LIN {X 0,Y 278.895,Z 532.06,A -85,B 0,C 180,E1 8838.94,E2 8838.94} C_VEL
LIN {X 0,Y 275.057,Z 524.837,A -85,B 0,C 180,E1 8835.829,E2 8835.829} C_VEL
LIN {X 0,Y 272.433,Z 520.123,A -85,B 0,C 180,E1 8833.269,E2 8833.269} C_VEL
LIN {X 0,Y 270.738,Z 517.123,A -85,B 0,C 180,E1 8831.296,E2 8831.296} C_VEL
LIN {X 0,Y 268.744,Z 513.445,A -85,B 0,C 180,E1 8828.352,E2 8828.352} C_VEL
LIN {X 0,Y 266.68,Z 509.32,A -85,B 0,C 180,E1 8823.018,E2 8823.018} C_VEL
LIN {X 0,Y 266.52,Z 508.712,A -85,B 0,C 180,E1 8821.944,E2 8821.944} C_VEL
LIN {X 0,Y 266.628,Z 508.877,A -85,B 0,C 180,E1 8817,E2 8817} C_VEL
LIN {X 0,Y 268.614,Z 513.288,A -85,B 0,C 180,E1 8811.447,E2 8811.447} C_VEL
LIN {X 0,Y 269.377,Z 514.72,A -85,B 0,C 180,E1 8810.179,E2 8810.179} C_VEL
LIN {X 0,Y 271.686,Z 518.794,A -85,B 0,C 180,E1 8807.145,E2 8807.145} C_VEL
LIN {X 0,Y 274.494,Z 523.834,A -85,B 0,C 180,E1 8804.265,E2 8804.265} C_VEL
LIN {X 0,Y 284.52,Z 539.001,A -85,B 0,C 180,E1 8797.161,E2 8797.161} C_VEL
LIN {X 0,Y 294.032,Z 548.26,A -85,B 0,C 180,E1 8792.575,E2 8792.575} C_VEL
LIN {X 0,Y 299.844,Z 552.837,A -85,B 0,C 180,E1 8790.22,E2 8790.22} C_VEL
LIN {X 0,Y 306.132,Z 557.593,A -85,B 0,C 180,E1 8787.514,E2 8787.514} C_VEL
LIN {X 0,Y 312.499,Z 562.998,A -85,B 0,C 180,E1 8784.512,E2 8784.512} C_VEL
LIN {X 0,Y 317.671,Z 567.158,A -85,B 0,C 180,E1 8781.808,E2 8781.808} C_VEL
LIN {X 0,Y 322.992,Z 572.197,A -85,B 0,C 180,E1 8778.644,E2 8778.644} C_VEL
LIN {X 0,Y 326.237,Z 574.988,A -85,B 0,C 180,E1 8776.659,E2 8776.659} C_VEL
LIN {X 0,Y 331.205,Z 579.653,A -85,B 0,C 180,E1 8773.494,E2 8773.494} C_VEL
LIN {X 0,Y 334.739,Z 582.505,A -85,B 0,C 180,E1 8771.19,E2 8771.19} C_VEL
LIN {X 0,Y 339.474,Z 587.061,A -85,B 0,C 180,E1 8767.893,E2 8767.893} C_VEL
LIN {X 0,Y 343.653,Z 590.222,A -85,B 0,C 180,E1 8764.886,E2 8764.886} C_VEL
LIN {X 0,Y 347.419,Z 593.994,A -85,B 0,C 180,E1 8761.917,E2 8761.917} C_VEL
LIN {X 0,Y 351.248,Z 596.825,A -85,B 0,C 180,E1 8758.755,E2 8758.755} C_VEL
LIN {X 0,Y 353.096,Z 598.088,A -85,B 0,C 180,E1 8757.122,E2 8757.122} C_VEL
LIN {X 0,Y 356.171,Z 601.48,A -85,B 0,C 180,E1 8754.019,E2 8754.019} C_VEL
LIN {X 0,Y 359.21,Z 603.908,A -85,B 0,C 180,E1 8750.701,E2 8750.701} C_VEL
LIN {X 0,Y 361.941,Z 605.377,A -85,B 0,C 180,E1 8747.358,E2 8747.358} C_VEL
LIN {X 0,Y 363.254,Z 606.183,A -85,B 0,C 180,E1 8745.485,E2 8745.485} C_VEL
LIN {X 0,Y 365.032,Z 608.588,A -85,B 0,C 180,E1 8742.336,E2 8742.336} C_VEL
LIN {X 0,Y 366.44,Z 610.11,A -85,B 0,C 180,E1 8739.05,E2 8739.05} C_VEL
LIN {X 0,Y 367.523,Z 611.035,A -85,B 0,C 180,E1 8735.62,E2 8735.62} C_VEL
LIN {X 0,Y 368.125,Z 611.482,A -85,B 0,C 180,E1 8732.179,E2 8732.179} C_VEL
LIN {X 0,Y 368.163,Z 611.49,A -85,B 0,C 180,E1 8728.911,E2 8728.911} C_VEL
LIN {X 0,Y 367.82,Z 611.243,A -85,B 0,C 180,E1 8725.635,E2 8725.635} C_VEL
LIN {X 0,Y 366.897,Z 610.529,A -85,B 0,C 180,E1 8722.169,E2 8722.169} C_VEL
LIN {X 0,Y 365.612,Z 609.266,A -85,B 0,C 180,E1 8718.964,E2 8718.964} C_VEL
LIN {X 0,Y 364.032,Z 607.268,A -85,B 0,C 180,E1 8715.782,E2 8715.782} C_VEL
LIN {X 0,Y 362.594,Z 605.615,A -85,B 0,C 180,E1 8713.5,E2 8713.5} C_VEL
LIN {X 0,Y 359.86,Z 604.308,A -85,B 0,C 180,E1 8710.017,E2 8710.017} C_VEL
LIN {X 0,Y 356.901,Z 602.129,A -85,B 0,C 180,E1 8706.734,E2 8706.734} C_VEL
LIN {X 0,Y 353.792,Z 598.981,A -85,B 0,C 180,E1 8703.597,E2 8703.597} C_VEL
LIN {X 0,Y 352.164,Z 597.33,A -85,B 0,C 180,E1 8702.066,E2 8702.066} C_VEL
LIN {X 0,Y 348.411,Z 594.838,A -85,B 0,C 180,E1 8698.899,E2 8698.899} C_VEL
LIN {X 0,Y 344.448,Z 591.117,A -85,B 0,C 180,E1 8695.728,E2 8695.728} C_VEL
LIN {X 0,Y 342.485,Z 589.191,A -85,B 0,C 180,E1 8694.234,E2 8694.234} C_VEL
LIN {X 0,Y 338.18,Z 585.932,A -85,B 0,C 180,E1 8691.187,E2 8691.187} C_VEL
LIN {X 0,Y 333.157,Z 581.089,A -85,B 0,C 180,E1 8687.76,E2 8687.76} C_VEL
LIN {X 0,Y 328.196,Z 577.001,A -85,B 0,C 180,E1 8684.579,E2 8684.579} C_VEL
LIN {X 0,Y 324.234,Z 573.152,A -85,B 0,C 180,E1 8682.108,E2 8682.108} C_VEL
LIN {X 0,Y 319.076,Z 568.633,A -85,B 0,C 180,E1 8679.026,E2 8679.026} C_VEL
LIN {X 0,Y 315.336,Z 565.145,A -85,B 0,C 180,E1 8676.919,E2 8676.919} C_VEL
LIN {X 0,Y 309.925,Z 560.861,A -85,B 0,C 180,E1 8674.248,E2 8674.248} C_VEL
LIN {X 0,Y 305.541,Z 557.19,A -85,B 0,C 180,E1 8672.223,E2 8672.223} C_VEL
LIN {X 0,Y 298.76,Z 551.933,A -85,B 0,C 180,E1 8669.348,E2 8669.348} C_VEL
LIN {X 0,Y 287.991,Z 542.764,A -85,B 0,C 180,E1 8664.665,E2 8664.665} C_VEL
LIN {X 0,Y 280.024,Z 533.138,A -85,B 0,C 180,E1 8660.09,E2 8660.09} C_VEL
LIN {X 0,Y 273.336,Z 521.624,A -85,B 0,C 180,E1 8654.609,E2 8654.609} C_VEL
LIN {X 0,Y 270.651,Z 517.002,A -85,B 0,C 180,E1 8651.605,E2 8651.605} C_VEL
LIN {X 0,Y 268.746,Z 513.415,A -85,B 0,C 180,E1 8648.764,E2 8648.764} C_VEL
LIN {X 0,Y 266.64,Z 508.986,A -85,B 0,C 180,E1 8643.107,E2 8643.107} C_VEL
LIN {X 0,Y 266.486,Z 508.701,A -85,B 0,C 180,E1 8638.271,E2 8638.271} C_VEL
LIN {X 0,Y 266.665,Z 509.22,A -85,B 0,C 180,E1 8637.089,E2 8637.089} C_VEL
LIN {X 0,Y 268.613,Z 513.317,A -85,B 0,C 180,E1 8631.86,E2 8631.86} C_VEL
LIN {X 0,Y 269.377,Z 514.737,A -85,B 0,C 180,E1 8630.592,E2 8630.592} C_VEL
LIN {X 0,Y 271.784,Z 518.909,A -85,B 0,C 180,E1 8627.456,E2 8627.456} C_VEL
LIN {X 0,Y 274.273,Z 523.465,A -85,B 0,C 180,E1 8624.883,E2 8624.883} C_VEL
LIN {X 0,Y 277.465,Z 529.282,A -85,B 0,C 180,E1 8622.155,E2 8622.155} C_VEL
LIN {X 0,Y 280.369,Z 535.335,A -85,B 0,C 180,E1 8619.972,E2 8619.972} C_VEL
LIN {X 0,Y 281.017,Z 537.508,A -85,B 0,C 180,E1 8619.462,E2 8619.462} C_VEL
LIN {X 0,Y 271.138,Z 641.697,A -85,B 0,C 180,E1 8617.288,E2 8617.288} C_VEL
LIN {X 0,Y 267.223,Z 664.526,A -85,B 0,C 180,E1 8616.63,E2 8616.63} C_VEL
LIN {X 0,Y 263.041,Z 681.531,A -85,B 0,C 180,E1 8615.964,E2 8615.964} C_VEL
LIN {X 0,Y 257.934,Z 698.333,A -85,B 0,C 180,E1 8615.101,E2 8615.101} C_VEL
LIN {X 0,Y 250.339,Z 718.684,A -85,B 0,C 180,E1 8613.719,E2 8613.719} C_VEL
LIN {X 0,Y 243.385,Z 734.31,A -85,B 0,C 180,E1 8612.331,E2 8612.331} C_VEL
LIN {X 0,Y 235.714,Z 749.491,A -85,B 0,C 180,E1 8610.653,E2 8610.653} C_VEL
LIN {X 0,Y 225.819,Z 766.74,A -85,B 0,C 180,E1 8608.222,E2 8608.222} C_VEL
LIN {X 0,Y 216.717,Z 780.747,A -85,B 0,C 180,E1 8605.672,E2 8605.672} C_VEL
LIN {X 0,Y 208.118,Z 792.952,A -85,B 0,C 180,E1 8602.891,E2 8602.891} C_VEL
LIN {X 0,Y 197.528,Z 806.818,A -85,B 0,C 180,E1 8598.836,E2 8598.836} C_VEL
LIN {X 0,Y 188.815,Z 817.411,A -85,B 0,C 180,E1 8594.771,E2 8594.771} C_VEL
LIN {X 0,Y 185.36,Z 821.62,A -85,B 0,C 180,E1 8592.894,E2 8592.894} C_VEL
LIN {X 0,Y 181.356,Z 825.4,A -85,B 0,C 180,E1 8591.182,E2 8591.182} C_VEL
LIN {X 0,Y 168.049,Z 834.548,A -85,B 0,C 180,E1 8586.633,E2 8586.633} C_VEL
LIN {X 0,Y 165.072,Z 837.01,A -85,B 0,C 180,E1 8584.778,E2 8584.778} C_VEL
LIN {X 0,Y 159.783,Z 842.971,A -85,B 0,C 180,E1 8579.214,E2 8579.214} C_VEL
LIN {X 0,Y 155.155,Z 848.829,A -85,B 0,C 180,E1 8571.846,E2 8571.846} C_VEL
LIN {X 0,Y 152.714,Z 852.655,A -85,B 0,C 180,E1 8564.406,E2 8564.406} C_VEL
LIN {X 0,Y 152.039,Z 854.633,A -85,B 0,C 180,E1 8558.318,E2 8558.318} C_VEL
LIN {X 0,Y 152.004,Z 855.505,A -85,B 0,C 180,E1 8553.016,E2 8553.016} C_VEL
LIN {X 0,Y 152.02,Z 855.596,A -85,B 0,C 180,E1 8548.115,E2 8548.115} C_VEL
LIN {X 0,Y 152.021,Z 854.815,A -85,B 0,C 180,E1 8542.442,E2 8542.442} C_VEL
LIN {X 0,Y 152.575,Z 852.957,A -85,B 0,C 180,E1 8536.355,E2 8536.355} C_VEL
LIN {X 0,Y 154.388,Z 849.835,A -85,B 0,C 180,E1 8529.926,E2 8529.926} C_VEL
LIN {X 0,Y 158.437,Z 844.654,A -85,B 0,C 180,E1 8522.57,E2 8522.57} C_VEL
LIN {X 0,Y 164.428,Z 837.72,A -85,B 0,C 180,E1 8515.812,E2 8515.812} C_VEL
LIN {X 0,Y 171.11,Z 830.424,A -85,B 0,C 180,E1 8510.438,E2 8510.438} C_VEL
LIN {X 0,Y 180.588,Z 820.031,A -85,B 0,C 180,E1 8504.696,E2 8504.696} C_VEL
LIN {X 0,Y 189.382,Z 809.898,A -85,B 0,C 180,E1 8500.509,E2 8500.509} C_VEL
LIN {X 0,Y 198.041,Z 799.411,A -85,B 0,C 180,E1 8497.091,E2 8497.091} C_VEL
LIN {X 0,Y 208.739,Z 785.512,A -85,B 0,C 180,E1 8493.547,E2 8493.547} C_VEL
LIN {X 0,Y 218.699,Z 770.992,A -85,B 0,C 180,E1 8490.741,E2 8490.741} C_VEL
LIN {X 0,Y 227.256,Z 757.259,A -85,B 0,C 180,E1 8488.633,E2 8488.633} C_VEL
LIN {X 0,Y 236.91,Z 739.862,A -85,B 0,C 180,E1 8486.53,E2 8486.53} C_VEL
LIN {X 0,Y 244.849,Z 723.051,A -85,B 0,C 180,E1 8484.971,E2 8484.971} C_VEL
LIN {X 0,Y 251.35,Z 707.199,A -85,B 0,C 180,E1 8483.808,E2 8483.808} C_VEL
LIN {X 0,Y 257.973,Z 688.057,A -85,B 0,C 180,E1 8482.718,E2 8482.718} C_VEL
LIN {X 0,Y 263.191,Z 668.401,A -85,B 0,C 180,E1 8481.912,E2 8481.912} C_VEL
LIN {X 0,Y 266.733,Z 650.8,A -85,B 0,C 180,E1 8481.37,E2 8481.37} C_VEL
LIN {X 0,Y 269.745,Z 627.11,A -85,B 0,C 180,E1 8480.812,E2 8480.812} C_VEL
LIN {X 0,Y 277.893,Z 541.402,A -85,B 0,C 180,E1 8479.066,E2 8479.066} C_VEL
LIN {X 0,Y 274.668,Z 534.689,A -85,B 0,C 180,E1 8476.449,E2 8476.449} C_VEL
LIN {X 0,Y 271.145,Z 527.997,A -85,B 0,C 180,E1 8473.008,E2 8473.008} C_VEL
LIN {X 0,Y 269.338,Z 524.692,A -85,B 0,C 180,E1 8470.814,E2 8470.814} C_VEL
LIN {X 0,Y 267.512,Z 521.194,A -85,B 0,C 180,E1 8467.958,E2 8467.958} C_VEL
LIN {X 0,Y 265.619,Z 516.917,A -85,B 0,C 180,E1 8462.49,E2 8462.49} C_VEL
LIN {X 0,Y 265.6,Z 516.697,A -85,B 0,C 180,E1 8457.312,E2 8457.312} C_VEL
LIN {X 0,Y 267.514,Z 521.166,A -85,B 0,C 180,E1 8451.628,E2 8451.628} C_VEL
LIN {X 0,Y 270.26,Z 526.374,A -85,B 0,C 180,E1 8447.599,E2 8447.599} C_VEL
LIN {X 0,Y 272.833,Z 531.197,A -85,B 0,C 180,E1 8444.82,E2 8444.82} C_VEL
LIN {X 0,Y 282.543,Z 546.368,A -85,B 0,C 180,E1 8437.652,E2 8437.652} C_VEL
LIN {X 0,Y 292.072,Z 555.804,A -85,B 0,C 180,E1 8432.927,E2 8432.927} C_VEL
LIN {X 0,Y 299.552,Z 561.757,A -85,B 0,C 180,E1 8429.857,E2 8429.857} C_VEL
LIN {X 0,Y 306.439,Z 566.905,A -85,B 0,C 180,E1 8426.884,E2 8426.884} C_VEL
LIN {X 0,Y 312.333,Z 571.835,A -85,B 0,C 180,E1 8424.038,E2 8424.038} C_VEL
LIN {X 0,Y 316.143,Z 574.926,A -85,B 0,C 180,E1 8422.051,E2 8422.051} C_VEL
LIN {X 0,Y 321.379,Z 579.816,A -85,B 0,C 180,E1 8418.984,E2 8418.984} C_VEL
LIN {X 0,Y 324.796,Z 582.75,A -85,B 0,C 180,E1 8416.904,E2 8416.904} C_VEL
LIN {X 0,Y 329.814,Z 587.419,A -85,B 0,C 180,E1 8413.724,E2 8413.724} C_VEL
LIN {X 0,Y 333.493,Z 590.415,A -85,B 0,C 180,E1 8411.336,E2 8411.336} C_VEL
LIN {X 0,Y 338.248,Z 594.926,A -85,B 0,C 180,E1 8408.04,E2 8408.04} C_VEL
LIN {X 0,Y 342.443,Z 598.118,A -85,B 0,C 180,E1 8405.034,E2 8405.034} C_VEL
LIN {X 0,Y 346.371,Z 601.979,A -85,B 0,C 180,E1 8401.952,E2 8401.952} C_VEL
LIN {X 0,Y 350.368,Z 604.862,A -85,B 0,C 180,E1 8398.647,E2 8398.647} C_VEL
LIN {X 0,Y 352.084,Z 606.158,A -85,B 0,C 180,E1 8397.123,E2 8397.123} C_VEL
LIN {X 0,Y 355.313,Z 609.596,A -85,B 0,C 180,E1 8393.884,E2 8393.884} C_VEL
LIN {X 0,Y 358.324,Z 611.937,A -85,B 0,C 180,E1 8390.584,E2 8390.584} C_VEL
LIN {X 0,Y 361.059,Z 613.362,A -85,B 0,C 180,E1 8387.216,E2 8387.216} C_VEL
LIN {X 0,Y 362.242,Z 614.145,A -85,B 0,C 180,E1 8385.529,E2 8385.529} C_VEL
LIN {X 0,Y 364.026,Z 616.531,A -85,B 0,C 180,E1 8382.371,E2 8382.371} C_VEL
LIN {X 0,Y 365.451,Z 618.049,A -85,B 0,C 180,E1 8379.073,E2 8379.073} C_VEL
LIN {X 0,Y 366.544,Z 618.975,A -85,B 0,C 180,E1 8375.635,E2 8375.635} C_VEL
LIN {X 0,Y 367.15,Z 619.423,A -85,B 0,C 180,E1 8372.185,E2 8372.185} C_VEL
LIN {X 0,Y 367.186,Z 619.43,A -85,B 0,C 180,E1 8368.908,E2 8368.908} C_VEL
LIN {X 0,Y 366.838,Z 619.182,A -85,B 0,C 180,E1 8365.623,E2 8365.623} C_VEL
LIN {X 0,Y 365.952,Z 618.516,A -85,B 0,C 180,E1 8362.306,E2 8362.306} C_VEL
LIN {X 0,Y 364.628,Z 617.227,A -85,B 0,C 180,E1 8358.96,E2 8358.96} C_VEL
LIN {X 0,Y 363.031,Z 615.245,A -85,B 0,C 180,E1 8355.763,E2 8355.763} C_VEL
LIN {X 0,Y 361.57,Z 613.544,A -85,B 0,C 180,E1 8353.452,E2 8353.452} C_VEL
LIN {X 0,Y 358.972,Z 612.321,A -85,B 0,C 180,E1 8350.135,E2 8350.135} C_VEL
LIN {X 0,Y 356.011,Z 610.204,A -85,B 0,C 180,E1 8346.848,E2 8346.848} C_VEL
LIN {X 0,Y 352.767,Z 607.007,A -85,B 0,C 180,E1 8343.578,E2 8343.578} C_VEL
LIN {X 0,Y 351.056,Z 605.231,A -85,B 0,C 180,E1 8341.97,E2 8341.97} C_VEL
LIN {X 0,Y 347.231,Z 602.709,A -85,B 0,C 180,E1 8338.763,E2 8338.763} C_VEL
LIN {X 0,Y 343.157,Z 598.927,A -85,B 0,C 180,E1 8335.527,E2 8335.527} C_VEL
LIN {X 0,Y 340.974,Z 596.877,A -85,B 0,C 180,E1 8333.887,E2 8333.887} C_VEL
LIN {X 0,Y 336.485,Z 593.404,A -85,B 0,C 180,E1 8330.735,E2 8330.735} C_VEL
LIN {X 0,Y 331.805,Z 588.879,A -85,B 0,C 180,E1 8327.548,E2 8327.548} C_VEL
LIN {X 0,Y 326.77,Z 584.766,A -85,B 0,C 180,E1 8324.346,E2 8324.346} C_VEL
LIN {X 0,Y 322.635,Z 580.784,A -85,B 0,C 180,E1 8321.768,E2 8321.768} C_VEL
LIN {X 0,Y 317.419,Z 576.231,A -85,B 0,C 180,E1 8318.688,E2 8318.688} C_VEL
LIN {X 0,Y 313.764,Z 572.877,A -85,B 0,C 180,E1 8316.678,E2 8316.678} C_VEL
LIN {X 0,Y 308.135,Z 568.446,A -85,B 0,C 180,E1 8313.913,E2 8313.913} C_VEL
LIN {X 0,Y 303.304,Z 564.494,A -85,B 0,C 180,E1 8311.71,E2 8311.71} C_VEL
LIN {X 0,Y 296.567,Z 559.304,A -85,B 0,C 180,E1 8308.922,E2 8308.922} C_VEL
LIN {X 0,Y 286.028,Z 550.228,A -85,B 0,C 180,E1 8304.24,E2 8304.24} C_VEL
LIN {X 0,Y 278.095,Z 540.397,A -85,B 0,C 180,E1 8299.523,E2 8299.523} C_VEL
LIN {X 0,Y 271.724,Z 529.017,A -85,B 0,C 180,E1 8294.045,E2 8294.045} C_VEL
LIN {X 0,Y 269.337,Z 524.691,A -85,B 0,C 180,E1 8291.228,E2 8291.228} C_VEL
LIN {X 0,Y 267.514,Z 521.166,A -85,B 0,C 180,E1 8288.372,E2 8288.372} C_VEL
LIN {X 0,Y 265.545,Z 516.653,A -85,B 0,C 180,E1 8282.364,E2 8282.364} C_VEL
LIN {X 0,Y 265.619,Z 516.917,A -85,B 0,C 180,E1 8277.51,E2 8277.51} C_VEL
LIN {X 0,Y 267.512,Z 521.194,A -85,B 0,C 180,E1 8272.042,E2 8272.042} C_VEL
LIN {X 0,Y 270.337,Z 526.453,A -85,B 0,C 180,E1 8267.93,E2 8267.93} C_VEL
LIN {X 0,Y 272.936,Z 531.424,A -85,B 0,C 180,E1 8265.133,E2 8265.133} C_VEL
LIN {X 0,Y 276.109,Z 537.585,A -85,B 0,C 180,E1 8262.337,E2 8262.337} C_VEL
LIN {X 0,Y 277.894,Z 541.512,A -85,B 0,C 180,E1 8260.926,E2 8260.926} C_VEL
LIN {X 0,Y 268.116,Z 641.667,A -85,B 0,C 180,E1 8258.866,E2 8258.866} C_VEL
LIN {X 0,Y 264.072,Z 664.592,A -85,B 0,C 180,E1 8258.217,E2 8258.217} C_VEL
LIN {X 0,Y 259.921,Z 681.125,A -85,B 0,C 180,E1 8257.589,E2 8257.589} C_VEL
LIN {X 0,Y 255.021,Z 696.98,A -85,B 0,C 180,E1 8256.805,E2 8256.805} C_VEL
LIN {X 0,Y 248.096,Z 715.668,A -85,B 0,C 180,E1 8255.613,E2 8255.613} C_VEL
LIN {X 0,Y 240.061,Z 733.408,A -85,B 0,C 180,E1 8254.108,E2 8254.108} C_VEL
LIN {X 0,Y 232.621,Z 747.828,A -85,B 0,C 180,E1 8252.568,E2 8252.568} C_VEL
LIN {X 0,Y 223.504,Z 763.57,A -85,B 0,C 180,E1 8250.468,E2 8250.468} C_VEL
LIN {X 0,Y 212.932,Z 779.505,A -85,B 0,C 180,E1 8247.693,E2 8247.693} C_VEL
LIN {X 0,Y 203.957,Z 791.818,A -85,B 0,C 180,E1 8244.951,E2 8244.951} C_VEL
LIN {X 0,Y 193.631,Z 804.96,A -85,B 0,C 180,E1 8241.233,E2 8241.233} C_VEL
LIN {X 0,Y 183.632,Z 816.547,A -85,B 0,C 180,E1 8236.853,E2 8236.853} C_VEL
LIN {X 0,Y 175.782,Z 825.3,A -85,B 0,C 180,E1 8232.599,E2 8232.599} C_VEL
LIN {X 0,Y 167.551,Z 834.392,A -85,B 0,C 180,E1 8226.885,E2 8226.885} C_VEL
LIN {X 0,Y 165.072,Z 837.01,A -85,B 0,C 180,E1 8224.778,E2 8224.778} C_VEL
LIN {X 0,Y 161.674,Z 839.89,A -85,B 0,C 180,E1 8222.527,E2 8222.527} C_VEL
LIN {X 0,Y 150.726,Z 845.91,A -85,B 0,C 180,E1 8216.73,E2 8216.73} C_VEL
LIN {X 0,Y 148.111,Z 847.909,A -85,B 0,C 180,E1 8214.037,E2 8214.037} C_VEL
LIN {X 0,Y 144.945,Z 852.263,A -85,B 0,C 180,E1 8205.606,E2 8205.606} C_VEL
LIN {X 0,Y 144.077,Z 854.304,A -85,B 0,C 180,E1 8199.184,E2 8199.184} C_VEL
LIN {X 0,Y 143.999,Z 855.237,A -85,B 0,C 180,E1 8193.583,E2 8193.583} C_VEL
LIN {X 0,Y 144.027,Z 855.389,A -85,B 0,C 180,E1 8188.409,E2 8188.409} C_VEL
LIN {X 0,Y 144.023,Z 854.668,A -85,B 0,C 180,E1 8182.421,E2 8182.421} C_VEL
LIN {X 0,Y 144.62,Z 852.868,A -85,B 0,C 180,E1 8175.997,E2 8175.997} C_VEL
LIN {X 0,Y 146.602,Z 849.772,A -85,B 0,C 180,E1 8169.163,E2 8169.163} C_VEL
LIN {X 0,Y 150.925,Z 844.72,A -85,B 0,C 180,E1 8161.512,E2 8161.512} C_VEL
LIN {X 0,Y 157.539,Z 837.642,A -85,B 0,C 180,E1 8154.276,E2 8154.276} C_VEL
LIN {X 0,Y 164.384,Z 830.652,A -85,B 0,C 180,E1 8148.937,E2 8148.937} C_VEL
LIN {X 0,Y 173.581,Z 821.245,A -85,B 0,C 180,E1 8143.468,E2 8143.468} C_VEL
LIN {X 0,Y 183.673,Z 810.21,A -85,B 0,C 180,E1 8138.772,E2 8138.772} C_VEL
LIN {X 0,Y 192.546,Z 799.963,A -85,B 0,C 180,E1 8135.388,E2 8135.388} C_VEL
LIN {X 0,Y 202.909,Z 787.117,A -85,B 0,C 180,E1 8132.057,E2 8132.057} C_VEL
LIN {X 0,Y 213.899,Z 771.874,A -85,B 0,C 180,E1 8129.062,E2 8129.062} C_VEL
LIN {X 0,Y 222.712,Z 758.259,A -85,B 0,C 180,E1 8126.975,E2 8126.975} C_VEL
LIN {X 0,Y 231.396,Z 743.318,A -85,B 0,C 180,E1 8125.147,E2 8125.147} C_VEL
LIN {X 0,Y 240.729,Z 724.655,A -85,B 0,C 180,E1 8123.381,E2 8123.381} C_VEL
LIN {X 0,Y 247.369,Z 709.087,A -85,B 0,C 180,E1 8122.244,E2 8122.244} C_VEL
LIN {X 0,Y 253.321,Z 692.741,A -85,B 0,C 180,E1 8121.301,E2 8121.301} C_VEL
LIN {X 0,Y 259.399,Z 672.025,A -85,B 0,C 180,E1 8120.405,E2 8120.405} C_VEL
LIN {X 0,Y 263.411,Z 653.366,A -85,B 0,C 180,E1 8119.824,E2 8119.824} C_VEL
LIN {X 0,Y 266.081,Z 635.287,A -85,B 0,C 180,E1 8119.381,E2 8119.381} C_VEL
LIN {X 0,Y 274.883,Z 546.094,A -85,B 0,C 180,E1 8117.58,E2 8117.58} C_VEL
LIN {X 0,Y 271.501,Z 539.175,A -85,B 0,C 180,E1 8114.511,E2 8114.511} C_VEL
LIN {X 0,Y 268.909,Z 533.998,A -85,B 0,C 180,E1 8111.591,E2 8111.591} C_VEL
LIN {X 0,Y 266.292,Z 528.944,A -85,B 0,C 180,E1 8107.56,E2 8107.56} C_VEL
LIN {X 0,Y 264.537,Z 524.582,A -85,B 0,C 180,E1 8101.742,E2 8101.742} C_VEL
LIN {X 0,Y 264.606,Z 524.804,A -85,B 0,C 180,E1 8097.302,E2 8097.302} C_VEL
LIN {X 0,Y 266.7,Z 529.664,A -85,B 0,C 180,E1 8091.277,E2 8091.277} C_VEL
LIN {X 0,Y 268.901,Z 534.069,A -85,B 0,C 180,E1 8087.992,E2 8087.992} C_VEL
LIN {X 0,Y 271.611,Z 539.341,A -85,B 0,C 180,E1 8084.969,E2 8084.969} C_VEL
LIN {X 0,Y 280.586,Z 553.734,A -85,B 0,C 180,E1 8078.149,E2 8078.149} C_VEL
LIN {X 0,Y 290.123,Z 563.348,A -85,B 0,C 180,E1 8073.284,E2 8073.284} C_VEL
LIN {X 0,Y 299.893,Z 571.038,A -85,B 0,C 180,E1 8069.23,E2 8069.23} C_VEL
LIN {X 0,Y 304.96,Z 574.839,A -85,B 0,C 180,E1 8067.039,E2 8067.039} C_VEL
LIN {X 0,Y 310.954,Z 579.702,A -85,B 0,C 180,E1 8064.195,E2 8064.195} C_VEL
LIN {X 0,Y 314.779,Z 582.857,A -85,B 0,C 180,E1 8062.204,E2 8062.204} C_VEL
LIN {X 0,Y 320.154,Z 587.745,A -85,B 0,C 180,E1 8059.091,E2 8059.091} C_VEL
LIN {X 0,Y 323.405,Z 590.571,A -85,B 0,C 180,E1 8057.113,E2 8057.113} C_VEL
LIN {X 0,Y 328.428,Z 595.184,A -85,B 0,C 180,E1 8053.955,E2 8053.955} C_VEL
LIN {X 0,Y 332.099,Z 598.164,A -85,B 0,C 180,E1 8051.584,E2 8051.584} C_VEL
LIN {X 0,Y 336.809,Z 602.61,A -85,B 0,C 180,E1 8048.347,E2 8048.347} C_VEL
LIN {X 0,Y 341.134,Z 605.891,A -85,B 0,C 180,E1 8045.267,E2 8045.267} C_VEL
LIN {X 0,Y 345.186,Z 609.843,A -85,B 0,C 180,E1 8042.102,E2 8042.102} C_VEL
LIN {X 0,Y 349.16,Z 612.707,A -85,B 0,C 180,E1 8038.827,E2 8038.827} C_VEL
LIN {X 0,Y 350.902,Z 614.029,A -85,B 0,C 180,E1 8037.274,E2 8037.274} C_VEL
LIN {X 0,Y 354.015,Z 617.333,A -85,B 0,C 180,E1 8034.174,E2 8034.174} C_VEL
LIN {X 0,Y 357.148,Z 619.775,A -85,B 0,C 180,E1 8030.794,E2 8030.794} C_VEL
LIN {X 0,Y 359.903,Z 621.234,A -85,B 0,C 180,E1 8027.459,E2 8027.459} C_VEL
LIN {X 0,Y 361.209,Z 622.074,A -85,B 0,C 180,E1 8025.612,E2 8025.612} C_VEL
LIN {X 0,Y 363.02,Z 624.473,A -85,B 0,C 180,E1 8022.405,E2 8022.405} C_VEL
LIN {X 0,Y 364.439,Z 625.97,A -85,B 0,C 180,E1 8019.156,E2 8019.156} C_VEL
LIN {X 0,Y 365.537,Z 626.883,A -85,B 0,C 180,E1 8015.808,E2 8015.808} C_VEL
LIN {X 0,Y 366.126,Z 627.328,A -85,B 0,C 180,E1 8012.504,E2 8012.504} C_VEL
LIN {X 0,Y 366.216,Z 627.381,A -85,B 0,C 180,E1 8009.061,E2 8009.061} C_VEL
LIN {X 0,Y 365.893,Z 627.139,A -85,B 0,C 180,E1 8005.733,E2 8005.733} C_VEL
LIN {X 0,Y 365.009,Z 626.499,A -85,B 0,C 180,E1 8002.445,E2 8002.445} C_VEL
LIN {X 0,Y 363.695,Z 625.245,A -85,B 0,C 180,E1 7999.065,E2 7999.065} C_VEL
LIN {X 0,Y 362.049,Z 623.242,A -85,B 0,C 180,E1 7995.772,E2 7995.772} C_VEL
LIN {X 0,Y 360.546,Z 621.473,A -85,B 0,C 180,E1 7993.404,E2 7993.404} C_VEL
LIN {X 0,Y 357.938,Z 620.246,A -85,B 0,C 180,E1 7990.075,E2 7990.075} C_VEL
LIN {X 0,Y 354.871,Z 618.058,A -85,B 0,C 180,E1 7986.682,E2 7986.682} C_VEL
LIN {X 0,Y 351.675,Z 614.949,A -85,B 0,C 180,E1 7983.49,E2 7983.49} C_VEL
LIN {X 0,Y 349.716,Z 613.015,A -85,B 0,C 180,E1 7981.667,E2 7981.667} C_VEL
LIN {X 0,Y 345.836,Z 610.404,A -85,B 0,C 180,E1 7978.447,E2 7978.447} C_VEL
LIN {X 0,Y 341.728,Z 606.579,A -85,B 0,C 180,E1 7975.213,E2 7975.213} C_VEL
LIN {X 0,Y 339.736,Z 604.724,A -85,B 0,C 180,E1 7973.727,E2 7973.727} C_VEL
LIN {X 0,Y 335.2,Z 601.239,A -85,B 0,C 180,E1 7970.555,E2 7970.555} C_VEL
LIN {X 0,Y 330.273,Z 596.544,A -85,B 0,C 180,E1 7967.219,E2 7967.219} C_VEL
LIN {X 0,Y 325.137,Z 592.331,A -85,B 0,C 180,E1 7963.981,E2 7963.981} C_VEL
LIN {X 0,Y 321.185,Z 588.529,A -85,B 0,C 180,E1 7961.521,E2 7961.521} C_VEL
LIN {X 0,Y 315.938,Z 583.988,A -85,B 0,C 180,E1 7958.439,E2 7958.439} C_VEL
LIN {X 0,Y 312.015,Z 580.484,A -85,B 0,C 180,E1 7956.346,E2 7956.346} C_VEL
LIN {X 0,Y 306.139,Z 575.864,A -85,B 0,C 180,E1 7953.489,E2 7953.489} C_VEL
LIN {X 0,Y 301.371,Z 572.062,A -85,B 0,C 180,E1 7951.379,E2 7951.379} C_VEL
LIN {X 0,Y 294.58,Z 566.858,A -85,B 0,C 180,E1 7948.581,E2 7948.581} C_VEL
LIN {X 0,Y 283.992,Z 557.591,A -85,B 0,C 180,E1 7943.762,E2 7943.762} C_VEL
LIN {X 0,Y 276.194,Z 547.655,A -85,B 0,C 180,E1 7938.949,E2 7938.949} C_VEL
LIN {X 0,Y 270.237,Z 536.562,A -85,B 0,C 180,E1 7933.578,E2 7933.578} C_VEL
LIN {X 0,Y 267.957,Z 532.259,A -85,B 0,C 180,E1 7930.742,E2 7930.742} C_VEL
LIN {X 0,Y 266.295,Z 528.914,A -85,B 0,C 180,E1 7927.976,E2 7927.976} C_VEL
LIN {X 0,Y 264.537,Z 524.576,A -85,B 0,C 180,E1 7922.157,E2 7922.157} C_VEL
LIN {X 0,Y 264.604,Z 524.819,A -85,B 0,C 180,E1 7917.717,E2 7917.717} C_VEL
LIN {X 0,Y 266.413,Z 529.072,A -85,B 0,C 180,E1 7912.226,E2 7912.226} C_VEL
LIN {X 0,Y 268.991,Z 534.175,A -85,B 0,C 180,E1 7908.304,E2 7908.304} C_VEL
LIN {X 0,Y 271.606,Z 539.367,A -85,B 0,C 180,E1 7905.386,E2 7905.386} C_VEL
LIN {X 0,Y 274.891,Z 546.109,A -85,B 0,C 180,E1 7902.414,E2 7902.414} C_VEL
LIN {X 0,Y 265.328,Z 641.44,A -85,B 0,C 180,E1 7900.482,E2 7900.482} C_VEL
LIN {X 0,Y 261.219,Z 664.273,A -85,B 0,C 180,E1 7899.855,E2 7899.855} C_VEL
LIN {X 0,Y 256.896,Z 681.129,A -85,B 0,C 180,E1 7899.235,E2 7899.235} C_VEL
LIN {X 0,Y 251.581,Z 697.858,A -85,B 0,C 180,E1 7898.428,E2 7898.428} C_VEL
LIN {X 0,Y 243.623,Z 718.207,A -85,B 0,C 180,E1 7897.124,E2 7897.124} C_VEL
LIN {X 0,Y 236.234,Z 733.976,A -85,B 0,C 180,E1 7895.794,E2 7895.794} C_VEL
LIN {X 0,Y 228.206,Z 749.012,A -85,B 0,C 180,E1 7894.204,E2 7894.204} C_VEL
LIN {X 0,Y 217.692,Z 766.259,A -85,B 0,C 180,E1 7891.864,E2 7891.864} C_VEL
LIN {X 0,Y 207.955,Z 780.265,A -85,B 0,C 180,E1 7889.386,E2 7889.386} C_VEL
LIN {X 0,Y 198.679,Z 792.469,A -85,B 0,C 180,E1 7886.655,E2 7886.655} C_VEL
LIN {X 0,Y 187.318,Z 806.144,A -85,B 0,C 180,E1 7882.684,E2 7882.684} C_VEL
LIN {X 0,Y 177.536,Z 816.926,A -85,B 0,C 180,E1 7878.505,E2 7878.505} C_VEL
LIN {X 0,Y 168.793,Z 826.145,A -85,B 0,C 180,E1 7873.871,E2 7873.871} C_VEL
LIN {X 0,Y 159.126,Z 836.032,A -85,B 0,C 180,E1 7867.099,E2 7867.099} C_VEL
LIN {X 0,Y 152.975,Z 842.397,A -85,B 0,C 180,E1 7861.079,E2 7861.079} C_VEL
LIN {X 0,Y 148.111,Z 847.909,A -85,B 0,C 180,E1 7854.037,E2 7854.037} C_VEL
LIN {X 0,Y 145.773,Z 849.751,A -85,B 0,C 180,E1 7851.241,E2 7851.241} C_VEL
LIN {X 0,Y 139.583,Z 852.307,A -85,B 0,C 180,E1 7846.042,E2 7846.042} C_VEL
LIN {X 0,Y 136.526,Z 853.559,A -85,B 0,C 180,E1 7842.084,E2 7842.084} C_VEL
LIN {X 0,Y 136.181,Z 853.858,A -85,B 0,C 180,E1 7840.69,E2 7840.69} C_VEL
LIN {X 0,Y 135.995,Z 854.969,A -85,B 0,C 180,E1 7834.216,E2 7834.216} C_VEL
LIN {X 0,Y 136.028,Z 855.153,A -85,B 0,C 180,E1 7828.315,E2 7828.315} C_VEL
LIN {X 0,Y 136.035,Z 854.43,A -85,B 0,C 180,E1 7821.973,E2 7821.973} C_VEL
LIN {X 0,Y 136.835,Z 852.476,A -85,B 0,C 180,E1 7814.747,E2 7814.747} C_VEL
LIN {X 0,Y 139.15,Z 849.352,A -85,B 0,C 180,E1 7807.616,E2 7807.616} C_VEL
LIN {X 0,Y 144.325,Z 843.889,A -85,B 0,C 180,E1 7799.237,E2 7799.237} C_VEL
LIN {X 0,Y 150.942,Z 837.399,A -85,B 0,C 180,E1 7792.454,E2 7792.454} C_VEL
LIN {X 0,Y 158.277,Z 830.409,A -85,B 0,C 180,E1 7786.982,E2 7786.982} C_VEL
LIN {X 0,Y 168.452,Z 820.588,A -85,B 0,C 180,E1 7781.228,E2 7781.228} C_VEL
LIN {X 0,Y 179.159,Z 809.422,A -85,B 0,C 180,E1 7776.523,E2 7776.523} C_VEL
LIN {X 0,Y 188.762,Z 798.771,A -85,B 0,C 180,E1 7773.078,E2 7773.078} C_VEL
LIN {X 0,Y 200.548,Z 784.529,A -85,B 0,C 180,E1 7769.545,E2 7769.545} C_VEL
LIN {X 0,Y 210.841,Z 770.51,A -85,B 0,C 180,E1 7766.936,E2 7766.936} C_VEL
LIN {X 0,Y 219.936,Z 756.778,A -85,B 0,C 180,E1 7764.916,E2 7764.916} C_VEL
LIN {X 0,Y 230.134,Z 739.384,A -85,B 0,C 180,E1 7762.921,E2 7762.921} C_VEL
LIN {X 0,Y 238.481,Z 722.574,A -85,B 0,C 180,E1 7761.451,E2 7761.451} C_VEL
LIN {X 0,Y 245.288,Z 706.723,A -85,B 0,C 180,E1 7760.362,E2 7760.362} C_VEL
LIN {X 0,Y 252.198,Z 687.582,A -85,B 0,C 180,E1 7759.345,E2 7759.345} C_VEL
LIN {X 0,Y 257.65,Z 667.846,A -85,B 0,C 180,E1 7758.596,E2 7758.596} C_VEL
LIN {X 0,Y 261.32,Z 650.282,A -85,B 0,C 180,E1 7758.089,E2 7758.089} C_VEL
LIN {X 0,Y 264.493,Z 626.381,A -85,B 0,C 180,E1 7757.555,E2 7757.555} C_VEL
LIN {X 0,Y 272.032,Z 551.115,A -85,B 0,C 180,E1 7756.071,E2 7756.071} C_VEL
LIN {X 0,Y 269.12,Z 544.927,A -85,B 0,C 180,E1 7753.107,E2 7753.107} C_VEL
LIN {X 0,Y 266.743,Z 540.068,A -85,B 0,C 180,E1 7750.047,E2 7750.047} C_VEL
LIN {X 0,Y 265.085,Z 536.691,A -85,B 0,C 180,E1 7747.159,E2 7747.159} C_VEL
LIN {X 0,Y 263.531,Z 532.515,A -85,B 0,C 180,E1 7741.531,E2 7741.531} C_VEL
LIN {X 0,Y 263.595,Z 532.71,A -85,B 0,C 180,E1 7737.51,E2 7737.51} C_VEL
LIN {X 0,Y 265.529,Z 537.508,A -85,B 0,C 180,E1 7731.565,E2 7731.565} C_VEL
LIN {X 0,Y 267.571,Z 541.792,A -85,B 0,C 180,E1 7728.369,E2 7728.369} C_VEL
LIN {X 0,Y 270.186,Z 547.087,A -85,B 0,C 180,E1 7725.326,E2 7725.326} C_VEL
LIN {X 0,Y 278.493,Z 560.915,A -85,B 0,C 180,E1 7718.75,E2 7718.75} C_VEL
LIN {X 0,Y 288.186,Z 570.892,A -85,B 0,C 180,E1 7713.646,E2 7713.646} C_VEL
LIN {X 0,Y 298.596,Z 579.047,A -85,B 0,C 180,E1 7709.305,E2 7709.305} C_VEL
LIN {X 0,Y 303.288,Z 582.592,A -85,B 0,C 180,E1 7707.284,E2 7707.284} C_VEL
LIN {X 0,Y 309.187,Z 587.299,A -85,B 0,C 180,E1 7704.529,E2 7704.529} C_VEL
LIN {X 0,Y 313.245,Z 590.618,A -85,B 0,C 180,E1 7702.448,E2 7702.448} C_VEL
LIN {X 0,Y 318.537,Z 595.368,A -85,B 0,C 180,E1 7699.428,E2 7699.428} C_VEL
LIN {X 0,Y 321.908,Z 598.272,A -85,B 0,C 180,E1 7697.396,E2 7697.396} C_VEL
LIN {X 0,Y 327.152,Z 603.045,A -85,B 0,C 180,E1 7694.108,E2 7694.108} C_VEL
LIN {X 0,Y 330.68,Z 605.915,A -85,B 0,C 180,E1 7691.829,E2 7691.829} C_VEL
LIN {X 0,Y 335.659,Z 610.537,A -85,B 0,C 180,E1 7688.442,E2 7688.442} C_VEL
LIN {X 0,Y 339.915,Z 613.789,A -85,B 0,C 180,E1 7685.412,E2 7685.412} C_VEL
LIN {X 0,Y 343.974,Z 617.699,A -85,B 0,C 180,E1 7682.254,E2 7682.254} C_VEL
LIN {X 0,Y 347.871,Z 620.513,A -85,B 0,C 180,E1 7679.06,E2 7679.06} C_VEL
LIN {X 0,Y 349.635,Z 621.803,A -85,B 0,C 180,E1 7677.504,E2 7677.504} C_VEL
LIN {X 0,Y 352.967,Z 625.284,A -85,B 0,C 180,E1 7674.224,E2 7674.224} C_VEL
LIN {X 0,Y 356.137,Z 627.722,A -85,B 0,C 180,E1 7670.819,E2 7670.819} C_VEL
LIN {X 0,Y 358.884,Z 629.163,A -85,B 0,C 180,E1 7667.511,E2 7667.511} C_VEL
LIN {X 0,Y 360.13,Z 629.924,A -85,B 0,C 180,E1 7665.788,E2 7665.788} C_VEL
LIN {X 0,Y 361.913,Z 632.322,A -85,B 0,C 180,E1 7662.606,E2 7662.606} C_VEL
LIN {X 0,Y 363.388,Z 633.861,A -85,B 0,C 180,E1 7659.342,E2 7659.342} C_VEL
LIN {X 0,Y 364.501,Z 634.753,A -85,B 0,C 180,E1 7656.141,E2 7656.141} C_VEL
LIN {X 0,Y 365.092,Z 635.229,A -85,B 0,C 180,E1 7652.825,E2 7652.825} C_VEL
LIN {X 0,Y 365.26,Z 635.352,A -85,B 0,C 180,E1 7649.373,E2 7649.373} C_VEL
LIN {X 0,Y 364.973,Z 635.125,A -85,B 0,C 180,E1 7646.073,E2 7646.073} C_VEL
LIN {X 0,Y 364.114,Z 634.513,A -85,B 0,C 180,E1 7642.743,E2 7642.743} C_VEL
LIN {X 0,Y 362.86,Z 633.355,A -85,B 0,C 180,E1 7639.361,E2 7639.361} C_VEL
LIN {X 0,Y 361.225,Z 631.454,A -85,B 0,C 180,E1 7636.066,E2 7636.066} C_VEL
LIN {X 0,Y 359.523,Z 629.402,A -85,B 0,C 180,E1 7633.355,E2 7633.355} C_VEL
LIN {X 0,Y 356.9,Z 628.17,A -85,B 0,C 180,E1 7630.015,E2 7630.015} C_VEL
LIN {X 0,Y 353.855,Z 626.019,A -85,B 0,C 180,E1 7626.655,E2 7626.655} C_VEL
LIN {X 0,Y 350.584,Z 622.889,A -85,B 0,C 180,E1 7623.401,E2 7623.401} C_VEL
LIN {X 0,Y 348.612,Z 620.916,A -85,B 0,C 180,E1 7621.57,E2 7621.57} C_VEL
LIN {X 0,Y 344.688,Z 618.297,A -85,B 0,C 180,E1 7618.33,E2 7618.33} C_VEL
LIN {X 0,Y 340.528,Z 614.478,A -85,B 0,C 180,E1 7615.072,E2 7615.072} C_VEL
LIN {X 0,Y 338.37,Z 612.486,A -85,B 0,C 180,E1 7613.471,E2 7613.471} C_VEL
LIN {X 0,Y 333.834,Z 608.994,A -85,B 0,C 180,E1 7610.313,E2 7610.313} C_VEL
LIN {X 0,Y 328.859,Z 604.296,A -85,B 0,C 180,E1 7606.973,E2 7606.973} C_VEL
LIN {X 0,Y 323.608,Z 599.987,A -85,B 0,C 180,E1 7603.672,E2 7603.672} C_VEL
LIN {X 0,Y 319.57,Z 596.156,A -85,B 0,C 180,E1 7601.18,E2 7601.18} C_VEL
LIN {X 0,Y 314.256,Z 591.586,A -85,B 0,C 180,E1 7598.102,E2 7598.102} C_VEL
LIN {X 0,Y 310.1,Z 587.961,A -85,B 0,C 180,E1 7595.919,E2 7595.919} C_VEL
LIN {X 0,Y 303.879,Z 583.107,A -85,B 0,C 180,E1 7592.981,E2 7592.981} C_VEL
LIN {X 0,Y 299.435,Z 579.628,A -85,B 0,C 180,E1 7591.045,E2 7591.045} C_VEL
LIN {X 0,Y 292.369,Z 574.223,A -85,B 0,C 180,E1 7588.148,E2 7588.148} C_VEL
LIN {X 0,Y 282.063,Z 565.053,A -85,B 0,C 180,E1 7583.325,E2 7583.325} C_VEL
LIN {X 0,Y 274.322,Z 554.913,A -85,B 0,C 180,E1 7578.367,E2 7578.367} C_VEL
LIN {X 0,Y 268.675,Z 543.952,A -85,B 0,C 180,E1 7573.001,E2 7573.001} C_VEL
LIN {X 0,Y 266.526,Z 539.7,A -85,B 0,C 180,E1 7570.145,E2 7570.145} C_VEL
LIN {X 0,Y 265.09,Z 536.659,A -85,B 0,C 180,E1 7567.576,E2 7567.576} C_VEL
LIN {X 0,Y 263.533,Z 532.5,A -85,B 0,C 180,E1 7561.947,E2 7561.947} C_VEL
LIN {X 0,Y 263.586,Z 532.618,A -85,B 0,C 180,E1 7558.034,E2 7558.034} C_VEL
LIN {X 0,Y 265.527,Z 537.52,A -85,B 0,C 180,E1 7551.982,E2 7551.982} C_VEL
LIN {X 0,Y 267.656,Z 541.894,A -85,B 0,C 180,E1 7548.681,E2 7548.681} C_VEL
LIN {X 0,Y 270.489,Z 547.695,A -85,B 0,C 180,E1 7545.433,E2 7545.433} C_VEL
LIN {X 0,Y 272.022,Z 551.376,A -85,B 0,C 180,E1 7543.912,E2 7543.912} C_VEL
LIN {X 0,Y 262.73,Z 641.41,A -85,B 0,C 180,E1 7542.127,E2 7542.127} C_VEL
LIN {X 0,Y 258.538,Z 664.151,A -85,B 0,C 180,E1 7541.521,E2 7541.521} C_VEL
LIN {X 0,Y 254.24,Z 680.619,A -85,B 0,C 180,E1 7540.94,E2 7540.94} C_VEL
LIN {X 0,Y 249.166,Z 696.375,A -85,B 0,C 180,E1 7540.216,E2 7540.216} C_VEL
LIN {X 0,Y 241.881,Z 715.192,A -85,B 0,C 180,E1 7539.096,E2 7539.096} C_VEL
LIN {X 0,Y 233.452,Z 732.93,A -85,B 0,C 180,E1 7537.681,E2 7537.681} C_VEL
LIN {X 0,Y 225.392,Z 747.732,A -85,B 0,C 180,E1 7536.181,E2 7536.181} C_VEL
LIN {X 0,Y 215.166,Z 764.326,A -85,B 0,C 180,E1 7534.047,E2 7534.047} C_VEL
LIN {X 0,Y 204.305,Z 779.524,A -85,B 0,C 180,E1 7531.455,E2 7531.455} C_VEL
LIN {X 0,Y 195.031,Z 791.335,A -85,B 0,C 180,E1 7528.884,E2 7528.884} C_VEL
LIN {X 0,Y 183.814,Z 804.476,A -85,B 0,C 180,E1 7525.219,E2 7525.219} C_VEL
LIN {X 0,Y 172.821,Z 816.062,A -85,B 0,C 180,E1 7520.826,E2 7520.826} C_VEL
LIN {X 0,Y 163.931,Z 824.943,A -85,B 0,C 180,E1 7516.415,E2 7516.415} C_VEL
LIN {X 0,Y 154.447,Z 834.168,A -85,B 0,C 180,E1 7510.343,E2 7510.343} C_VEL
LIN {X 0,Y 146.705,Z 841.475,A -85,B 0,C 180,E1 7503.507,E2 7503.507} C_VEL
LIN {X 0,Y 141.554,Z 846.667,A -85,B 0,C 180,E1 7496.875,E2 7496.875} C_VEL
LIN {X 0,Y 137.716,Z 851.25,A -85,B 0,C 180,E1 7488.629,E2 7488.629} C_VEL
LIN {X 0,Y 136.181,Z 853.858,A -85,B 0,C 180,E1 7480.69,E2 7480.69} C_VEL
LIN {X 0,Y 135.133,Z 854.509,A -85,B 0,C 180,E1 7477.688,E2 7477.688} C_VEL
LIN {X 0,Y 132.141,Z 854.909,A -85,B 0,C 180,E1 7473.571,E2 7473.571} C_VEL
LIN {X 0,Y 128.336,Z 854.906,A -85,B 0,C 180,E1 7467.546,E2 7467.546} C_VEL
LIN {X 0,Y 127.995,Z 854.732,A -85,B 0,C 180,E1 7465.525,E2 7465.525} C_VEL
LIN {X 0,Y 128.318,Z 853.459,A -85,B 0,C 180,E1 7457.855,E2 7457.855} C_VEL
LIN {X 0,Y 130.668,Z 850.169,A -85,B 0,C 180,E1 7448.452,E2 7448.452} C_VEL
LIN {X 0,Y 134.574,Z 846.151,A -85,B 0,C 180,E1 7441.124,E2 7441.124} C_VEL
LIN {X 0,Y 140.316,Z 840.895,A -85,B 0,C 180,E1 7434.247,E2 7434.247} C_VEL
LIN {X 0,Y 149.772,Z 832.524,A -85,B 0,C 180,E1 7426.56,E2 7426.56} C_VEL
LIN {X 0,Y 158.516,Z 824.571,A -85,B 0,C 180,E1 7421.359,E2 7421.359} C_VEL
LIN {X 0,Y 167.757,Z 815.82,A -85,B 0,C 180,E1 7417,E2 7417} C_VEL
LIN {X 0,Y 179.268,Z 804.234,A -85,B 0,C 180,E1 7412.63,E2 7412.63} C_VEL
LIN {X 0,Y 190.939,Z 791.094,A -85,B 0,C 180,E1 7409.017,E2 7409.017} C_VEL
LIN {X 0,Y 200.539,Z 779.283,A -85,B 0,C 180,E1 7406.5,E2 7406.5} C_VEL
LIN {X 0,Y 211.777,Z 764.025,A -85,B 0,C 180,E1 7403.967,E2 7403.967} C_VEL
LIN {X 0,Y 222.051,Z 747.821,A -85,B 0,C 180,E1 7401.943,E2 7401.943} C_VEL
LIN {X 0,Y 230.076,Z 733.498,A -85,B 0,C 180,E1 7400.531,E2 7400.531} C_VEL
LIN {X 0,Y 238.251,Z 716.809,A -85,B 0,C 180,E1 7399.227,E2 7399.227} C_VEL
LIN {X 0,Y 246.119,Z 697.382,A -85,B 0,C 180,E1 7398.085,E2 7398.085} C_VEL
LIN {X 0,Y 251.579,Z 680.887,A -85,B 0,C 180,E1 7397.351,E2 7397.351} C_VEL
LIN {X 0,Y 256.331,Z 662.998,A -85,B 0,C 180,E1 7396.748,E2 7396.748} C_VEL
LIN {X 0,Y 260.417,Z 640.772,A -85,B 0,C 180,E1 7396.184,E2 7396.184} C_VEL
LIN {X 0,Y 269.372,Z 556.284,A -85,B 0,C 180,E1 7394.546,E2 7394.546} C_VEL
LIN {X 0,Y 266.566,Z 550.123,A -85,B 0,C 180,E1 7391.256,E2 7391.256} C_VEL
LIN {X 0,Y 265.188,Z 547.262,A -85,B 0,C 180,E1 7389.23,E2 7389.23} C_VEL
LIN {X 0,Y 263.998,Z 544.569,A -85,B 0,C 180,E1 7386.97,E2 7386.97} C_VEL
LIN {X 0,Y 262.556,Z 540.455,A -85,B 0,C 180,E1 7381.537,E2 7381.537} C_VEL
LIN {X 0,Y 262.594,Z 540.712,A -85,B 0,C 180,E1 7377.609,E2 7377.609} C_VEL
LIN {X 0,Y 264.365,Z 545.349,A -85,B 0,C 180,E1 7371.856,E2 7371.856} C_VEL
LIN {X 0,Y 266.252,Z 549.514,A -85,B 0,C 180,E1 7368.75,E2 7368.75} C_VEL
LIN {X 0,Y 268.669,Z 554.676,A -85,B 0,C 180,E1 7365.792,E2 7365.792} C_VEL
LIN {X 0,Y 276.584,Z 568.28,A -85,B 0,C 180,E1 7359.262,E2 7359.262} C_VEL
LIN {X 0,Y 286.26,Z 578.436,A -85,B 0,C 180,E1 7354.013,E2 7354.013} C_VEL
LIN {X 0,Y 297.3,Z 587.051,A -85,B 0,C 180,E1 7349.381,E2 7349.381} C_VEL
LIN {X 0,Y 302.405,Z 591.016,A -85,B 0,C 180,E1 7347.176,E2 7347.176} C_VEL
LIN {X 0,Y 308.505,Z 595.688,A -85,B 0,C 180,E1 7344.325,E2 7344.325} C_VEL
LIN {X 0,Y 313.575,Z 600.112,A -85,B 0,C 180,E1 7341.684,E2 7341.684} C_VEL
LIN {X 0,Y 318.907,Z 604.472,A -85,B 0,C 180,E1 7338.597,E2 7338.597} C_VEL
LIN {X 0,Y 324.49,Z 609.803,A -85,B 0,C 180,E1 7335.128,E2 7335.128} C_VEL
LIN {X 0,Y 329.266,Z 613.665,A -85,B 0,C 180,E1 7332.075,E2 7332.075} C_VEL
LIN {X 0,Y 334.257,Z 618.283,A -85,B 0,C 180,E1 7328.69,E2 7328.69} C_VEL
LIN {X 0,Y 338.496,Z 621.48,A -85,B 0,C 180,E1 7325.697,E2 7325.697} C_VEL
LIN {X 0,Y 342.679,Z 625.489,A -85,B 0,C 180,E1 7322.47,E2 7322.47} C_VEL
LIN {X 0,Y 346.737,Z 628.407,A -85,B 0,C 180,E1 7319.164,E2 7319.164} C_VEL
LIN {X 0,Y 348.526,Z 629.757,A -85,B 0,C 180,E1 7317.591,E2 7317.591} C_VEL
LIN {X 0,Y 351.943,Z 633.257,A -85,B 0,C 180,E1 7314.25,E2 7314.25} C_VEL
LIN {X 0,Y 355.186,Z 635.706,A -85,B 0,C 180,E1 7310.774,E2 7310.774} C_VEL
LIN {X 0,Y 357.985,Z 637.142,A -85,B 0,C 180,E1 7307.388,E2 7307.388} C_VEL
LIN {X 0,Y 359.21,Z 638.037,A -85,B 0,C 180,E1 7305.656,E2 7305.656} C_VEL
LIN {X 0,Y 361.008,Z 640.357,A -85,B 0,C 180,E1 7302.476,E2 7302.476} C_VEL
LIN {X 0,Y 362.46,Z 641.846,A -85,B 0,C 180,E1 7299.206,E2 7299.206} C_VEL
LIN {X 0,Y 363.58,Z 642.764,A -85,B 0,C 180,E1 7295.84,E2 7295.84} C_VEL
LIN {X 0,Y 364.168,Z 643.208,A -85,B 0,C 180,E1 7292.518,E2 7292.518} C_VEL
LIN {X 0,Y 364.272,Z 643.278,A -85,B 0,C 180,E1 7289.214,E2 7289.214} C_VEL
LIN {X 0,Y 363.972,Z 643.046,A -85,B 0,C 180,E1 7285.904,E2 7285.904} C_VEL
LIN {X 0,Y 363.086,Z 642.416,A -85,B 0,C 180,E1 7282.564,E2 7282.564} C_VEL
LIN {X 0,Y 361.779,Z 641.217,A -85,B 0,C 180,E1 7279.168,E2 7279.168} C_VEL
LIN {X 0,Y 360.132,Z 639.285,A -85,B 0,C 180,E1 7275.859,E2 7275.859} C_VEL
LIN {X 0,Y 358.5,Z 637.331,A -85,B 0,C 180,E1 7273.306,E2 7273.306} C_VEL
LIN {X 0,Y 355.851,Z 636.092,A -85,B 0,C 180,E1 7269.954,E2 7269.954} C_VEL
LIN {X 0,Y 352.839,Z 633.979,A -85,B 0,C 180,E1 7266.627,E2 7266.627} C_VEL
LIN {X 0,Y 349.494,Z 630.827,A -85,B 0,C 180,E1 7263.311,E2 7263.311} C_VEL
LIN {X 0,Y 347.39,Z 628.753,A -85,B 0,C 180,E1 7261.362,E2 7261.362} C_VEL
LIN {X 0,Y 343.508,Z 626.163,A -85,B 0,C 180,E1 7258.184,E2 7258.184} C_VEL
LIN {X 0,Y 339.33,Z 622.375,A -85,B 0,C 180,E1 7254.931,E2 7254.931} C_VEL
LIN {X 0,Y 336.961,Z 620.216,A -85,B 0,C 180,E1 7253.175,E2 7253.175} C_VEL
LIN {X 0,Y 332.216,Z 616.527,A -85,B 0,C 180,E1 7249.906,E2 7249.906} C_VEL
LIN {X 0,Y 327.275,Z 611.94,A -85,B 0,C 180,E1 7246.63,E2 7246.63} C_VEL
LIN {X 0,Y 322.192,Z 607.755,A -85,B 0,C 180,E1 7243.435,E2 7243.435} C_VEL
LIN {X 0,Y 317.947,Z 603.781,A -85,B 0,C 180,E1 7240.838,E2 7240.838} C_VEL
LIN {X 0,Y 312.375,Z 599.024,A -85,B 0,C 180,E1 7237.674,E2 7237.674} C_VEL
LIN {X 0,Y 308.319,Z 595.56,A -85,B 0,C 180,E1 7235.586,E2 7235.586} C_VEL
LIN {X 0,Y 302.208,Z 590.852,A -85,B 0,C 180,E1 7232.735,E2 7232.735} C_VEL
LIN {X 0,Y 297.3,Z 587.051,A -85,B 0,C 180,E1 7230.619,E2 7230.619} C_VEL
LIN {X 0,Y 289.339,Z 580.834,A -85,B 0,C 180,E1 7227.35,E2 7227.35} C_VEL
LIN {X 0,Y 280.493,Z 572.914,A -85,B 0,C 180,E1 7223.075,E2 7223.075} C_VEL
LIN {X 0,Y 272.54,Z 562.286,A -85,B 0,C 180,E1 7217.827,E2 7217.827} C_VEL
LIN {X 0,Y 267.141,Z 551.341,A -85,B 0,C 180,E1 7212.417,E2 7212.417} C_VEL
LIN {X 0,Y 265.19,Z 547.264,A -85,B 0,C 180,E1 7209.649,E2 7209.649} C_VEL
LIN {X 0,Y 264.004,Z 544.538,A -85,B 0,C 180,E1 7207.388,E2 7207.388} C_VEL
LIN {X 0,Y 262.532,Z 540.425,A -85,B 0,C 180,E1 7201.736,E2 7201.736} C_VEL
LIN {X 0,Y 262.593,Z 540.712,A -85,B 0,C 180,E1 7198.027,E2 7198.027} C_VEL
LIN {X 0,Y 264.368,Z 545.373,A -85,B 0,C 180,E1 7192.264,E2 7192.264} C_VEL
LIN {X 0,Y 266.333,Z 549.611,A -85,B 0,C 180,E1 7189.063,E2 7189.063} C_VEL
LIN {X 0,Y 269.004,Z 555.42,A -85,B 0,C 180,E1 7185.846,E2 7185.846} C_VEL
LIN {X 0,Y 269.353,Z 556.495,A -85,B 0,C 180,E1 7185.449,E2 7185.449} C_VEL
LIN {X 0,Y 260.379,Z 641.184,A -85,B 0,C 180,E1 7183.808,E2 7183.808} C_VEL
LIN {X 0,Y 256.107,Z 663.914,A -85,B 0,C 180,E1 7183.224,E2 7183.224} C_VEL
LIN {X 0,Y 251.586,Z 680.864,A -85,B 0,C 180,E1 7182.649,E2 7182.649} C_VEL
LIN {X 0,Y 246.119,Z 697.382,A -85,B 0,C 180,E1 7181.915,E2 7181.915} C_VEL
LIN {X 0,Y 237.816,Z 717.73,A -85,B 0,C 180,E1 7180.707,E2 7180.707} C_VEL
LIN {X 0,Y 230.076,Z 733.498,A -85,B 0,C 180,E1 7179.47,E2 7179.47} C_VEL
LIN {X 0,Y 221.879,Z 748.112,A -85,B 0,C 180,E1 7178.026,E2 7178.026} C_VEL
LIN {X 0,Y 210.92,Z 765.217,A -85,B 0,C 180,E1 7175.855,E2 7175.855} C_VEL
LIN {X 0,Y 200.539,Z 779.283,A -85,B 0,C 180,E1 7173.5,E2 7173.5} C_VEL
LIN {X 0,Y 190.939,Z 791.094,A -85,B 0,C 180,E1 7170.983,E2 7170.983} C_VEL
LIN {X 0,Y 179.268,Z 804.234,A -85,B 0,C 180,E1 7167.37,E2 7167.37} C_VEL
LIN {X 0,Y 167.595,Z 815.976,A -85,B 0,C 180,E1 7162.931,E2 7162.931} C_VEL
LIN {X 0,Y 157.934,Z 825.115,A -85,B 0,C 180,E1 7158.333,E2 7158.333} C_VEL
LIN {X 0,Y 147.786,Z 834.338,A -85,B 0,C 180,E1 7152.049,E2 7152.049} C_VEL
LIN {X 0,Y 139.548,Z 841.569,A -85,B 0,C 180,E1 7144.972,E2 7144.972} C_VEL
LIN {X 0,Y 134.019,Z 846.698,A -85,B 0,C 180,E1 7138.034,E2 7138.034} C_VEL
LIN {X 0,Y 129.725,Z 851.328,A -85,B 0,C 180,E1 7128.887,E2 7128.887} C_VEL
LIN {X 0,Y 128.162,Z 853.794,A -85,B 0,C 180,E1 7120.497,E2 7120.497} C_VEL
LIN {X 0,Y 127.999,Z 854.763,A -85,B 0,C 180,E1 7114.031,E2 7114.031} C_VEL
LIN {X 0,Y 128.029,Z 854.916,A -85,B 0,C 180,E1 7108.21,E2 7108.21} C_VEL
LIN {X 0,Y 127.995,Z 854.732,A -85,B 0,C 180,E1 7105.525,E2 7105.525} C_VEL
LIN {X 0,Y 127.173,Z 854.373,A -85,B 0,C 180,E1 7102.321,E2 7102.321} C_VEL
LIN {X 0,Y 124.076,Z 853.28,A -85,B 0,C 180,E1 7097.175,E2 7097.175} C_VEL
LIN {X 0,Y 121.906,Z 851.699,A -85,B 0,C 180,E1 7091.793,E2 7091.793} C_VEL
LIN {X 0,Y 122.183,Z 850.951,A -85,B 0,C 180,E1 7089.45,E2 7089.45} C_VEL
LIN {X 0,Y 126.942,Z 846.364,A -85,B 0,C 180,E1 7080.077,E2 7080.077} C_VEL
LIN {X 0,Y 133.092,Z 841.168,A -85,B 0,C 180,E1 7072.806,E2 7072.806} C_VEL
LIN {X 0,Y 142.314,Z 833.682,A -85,B 0,C 180,E1 7065.368,E2 7065.368} C_VEL
LIN {X 0,Y 152.596,Z 824.872,A -85,B 0,C 180,E1 7059.362,E2 7059.362} C_VEL
LIN {X 0,Y 162.274,Z 816.199,A -85,B 0,C 180,E1 7054.969,E2 7054.969} C_VEL
LIN {X 0,Y 173.521,Z 805.418,A -85,B 0,C 180,E1 7050.847,E2 7050.847} C_VEL
LIN {X 0,Y 186.336,Z 791.745,A -85,B 0,C 180,E1 7047.037,E2 7047.037} C_VEL
LIN {X 0,Y 196.914,Z 779.197,A -85,B 0,C 180,E1 7044.408,E2 7044.408} C_VEL
LIN {X 0,Y 208.156,Z 764.403,A -85,B 0,C 180,E1 7042.015,E2 7042.015} C_VEL
LIN {X 0,Y 219.151,Z 747.581,A -85,B 0,C 180,E1 7039.977,E2 7039.977} C_VEL
LIN {X 0,Y 227.366,Z 733.259,A -85,B 0,C 180,E1 7038.622,E2 7038.622} C_VEL
LIN {X 0,Y 235.718,Z 716.571,A -85,B 0,C 180,E1 7037.376,E2 7037.376} C_VEL
LIN {X 0,Y 243.741,Z 697.144,A -85,B 0,C 180,E1 7036.286,E2 7036.286} C_VEL
LIN {X 0,Y 249.156,Z 681.128,A -85,B 0,C 180,E1 7035.606,E2 7035.606} C_VEL
LIN {X 0,Y 253.992,Z 663.333,A -85,B 0,C 180,E1 7035.031,E2 7035.031} C_VEL
LIN {X 0,Y 258.268,Z 640.741,A -85,B 0,C 180,E1 7034.478,E2 7034.478} C_VEL
LIN {X 0,Y 266.512,Z 565.091,A -85,B 0,C 180,E1 7033.049,E2 7033.049} C_VEL
LIN {X 0,Y 266.851,Z 561.555,A -85,B 0,C 180,E1 7032.951,E2 7032.951} C_VEL
LIN {X 0,Y 264.475,Z 555.922,A -85,B 0,C 180,E1 7029.694,E2 7029.694} C_VEL
LIN {X 0,Y 262.811,Z 552.313,A -85,B 0,C 180,E1 7026.563,E2 7026.563} C_VEL
LIN {X 0,Y 261.554,Z 548.388,A -85,B 0,C 180,E1 7021.324,E2 7021.324} C_VEL
LIN {X 0,Y 261.588,Z 548.611,A -85,B 0,C 180,E1 7017.819,E2 7017.819} C_VEL
LIN {X 0,Y 263.161,Z 553.043,A -85,B 0,C 180,E1 7012.258,E2 7012.258} C_VEL
LIN {X 0,Y 264.874,Z 557.059,A -85,B 0,C 180,E1 7009.241,E2 7009.241} C_VEL
LIN {X 0,Y 267.079,Z 562.054,A -85,B 0,C 180,E1 7006.369,E2 7006.369} C_VEL
LIN {X 0,Y 274.848,Z 575.83,A -85,B 0,C 180,E1 6999.682,E2 6999.682} C_VEL
LIN {X 0,Y 284.15,Z 585.821,A -85,B 0,C 180,E1 6994.478,E2 6994.478} C_VEL
LIN {X 0,Y 296.005,Z 595.046,A -85,B 0,C 180,E1 6989.457,E2 6989.457} C_VEL
LIN {X 0,Y 303.28,Z 600.785,A -85,B 0,C 180,E1 6986.267,E2 6986.267} C_VEL
LIN {X 0,Y 309.453,Z 605.478,A -85,B 0,C 180,E1 6983.305,E2 6983.305} C_VEL
LIN {X 0,Y 314.664,Z 610.136,A -85,B 0,C 180,E1 6980.438,E2 6980.438} C_VEL
LIN {X 0,Y 318.806,Z 613.588,A -85,B 0,C 180,E1 6978.011,E2 6978.011} C_VEL
LIN {X 0,Y 324.139,Z 618.425,A -85,B 0,C 180,E1 6974.691,E2 6974.691} C_VEL
LIN {X 0,Y 327.845,Z 621.4,A -85,B 0,C 180,E1 6972.334,E2 6972.334} C_VEL
LIN {X 0,Y 332.955,Z 626.105,A -85,B 0,C 180,E1 6968.874,E2 6968.874} C_VEL
LIN {X 0,Y 337.26,Z 629.369,A -85,B 0,C 180,E1 6965.847,E2 6965.847} C_VEL
LIN {X 0,Y 341.498,Z 633.374,A -85,B 0,C 180,E1 6962.596,E2 6962.596} C_VEL
LIN {X 0,Y 345.603,Z 636.301,A -85,B 0,C 180,E1 6959.269,E2 6959.269} C_VEL
LIN {X 0,Y 347.398,Z 637.685,A -85,B 0,C 180,E1 6957.698,E2 6957.698} C_VEL
LIN {X 0,Y 350.787,Z 641.111,A -85,B 0,C 180,E1 6954.411,E2 6954.411} C_VEL
LIN {X 0,Y 353.986,Z 643.527,A -85,B 0,C 180,E1 6951.021,E2 6951.021} C_VEL
LIN {X 0,Y 356.847,Z 645.019,A -85,B 0,C 180,E1 6947.614,E2 6947.614} C_VEL
LIN {X 0,Y 358.107,Z 645.847,A -85,B 0,C 180,E1 6945.879,E2 6945.879} C_VEL
LIN {X 0,Y 359.902,Z 648.207,A -85,B 0,C 180,E1 6942.678,E2 6942.678} C_VEL
LIN {X 0,Y 361.411,Z 649.737,A -85,B 0,C 180,E1 6939.394,E2 6939.394} C_VEL
LIN {X 0,Y 362.537,Z 650.633,A -85,B 0,C 180,E1 6936.174,E2 6936.174} C_VEL
LIN {X 0,Y 363.135,Z 651.11,A -85,B 0,C 180,E1 6932.841,E2 6932.841} C_VEL
LIN {X 0,Y 363.307,Z 651.233,A -85,B 0,C 180,E1 6929.369,E2 6929.369} C_VEL
LIN {X 0,Y 363.021,Z 651.006,A -85,B 0,C 180,E1 6926.052,E2 6926.052} C_VEL
LIN {X 0,Y 362.148,Z 650.391,A -85,B 0,C 180,E1 6922.704,E2 6922.704} C_VEL
LIN {X 0,Y 360.864,Z 649.239,A -85,B 0,C 180,E1 6919.302,E2 6919.302} C_VEL
LIN {X 0,Y 359.221,Z 647.363,A -85,B 0,C 180,E1 6915.987,E2 6915.987} C_VEL
LIN {X 0,Y 357.344,Z 645.215,A -85,B 0,C 180,E1 6913.083,E2 6913.083} C_VEL
LIN {X 0,Y 354.63,Z 643.922,A -85,B 0,C 180,E1 6909.709,E2 6909.709} C_VEL
LIN {X 0,Y 351.578,Z 641.753,A -85,B 0,C 180,E1 6906.361,E2 6906.361} C_VEL
LIN {X 0,Y 348.206,Z 638.541,A -85,B 0,C 180,E1 6903.02,E2 6903.02} C_VEL
LIN {X 0,Y 346.044,Z 636.537,A -85,B 0,C 180,E1 6901.08,E2 6901.08} C_VEL
LIN {X 0,Y 342.109,Z 633.856,A -85,B 0,C 180,E1 6897.866,E2 6897.866} C_VEL
LIN {X 0,Y 337.793,Z 629.924,A -85,B 0,C 180,E1 6894.54,E2 6894.54} C_VEL
LIN {X 0,Y 335.624,Z 628.009,A -85,B 0,C 180,E1 6892.96,E2 6892.96} C_VEL
LIN {X 0,Y 330.886,Z 624.341,A -85,B 0,C 180,E1 6889.711,E2 6889.711} C_VEL
LIN {X 0,Y 325.856,Z 619.691,A -85,B 0,C 180,E1 6886.382,E2 6886.382} C_VEL
LIN {X 0,Y 320.667,Z 615.44,A -85,B 0,C 180,E1 6883.147,E2 6883.147} C_VEL
LIN {X 0,Y 316.32,Z 611.405,A -85,B 0,C 180,E1 6880.495,E2 6880.495} C_VEL
LIN {X 0,Y 310.987,Z 606.935,A -85,B 0,C 180,E1 6877.523,E2 6877.523} C_VEL
LIN {X 0,Y 306.713,Z 603.288,A -85,B 0,C 180,E1 6875.342,E2 6875.342} C_VEL
LIN {X 0,Y 300.142,Z 598.259,A -85,B 0,C 180,E1 6872.309,E2 6872.309} C_VEL
LIN {X 0,Y 294.907,Z 594.315,A -85,B 0,C 180,E1 6870.106,E2 6870.106} C_VEL
LIN {X 0,Y 278.844,Z 580.668,A -85,B 0,C 180,E1 6862.773,E2 6862.773} C_VEL
LIN {X 0,Y 270.782,Z 569.658,A -85,B 0,C 180,E1 6857.281,E2 6857.281} C_VEL
LIN {X 0,Y 265.717,Z 558.885,A -85,B 0,C 180,E1 6851.934,E2 6851.934} C_VEL
LIN {X 0,Y 263.938,Z 554.953,A -85,B 0,C 180,E1 6849.255,E2 6849.255} C_VEL
LIN {X 0,Y 262.818,Z 552.28,A -85,B 0,C 180,E1 6846.982,E2 6846.982} C_VEL
LIN {X 0,Y 261.557,Z 548.366,A -85,B 0,C 180,E1 6841.743,E2 6841.743} C_VEL
LIN {X 0,Y 261.588,Z 548.608,A -85,B 0,C 180,E1 6838.238,E2 6838.238} C_VEL
LIN {X 0,Y 263.206,Z 553.193,A -85,B 0,C 180,E1 6832.57,E2 6832.57} C_VEL
LIN {X 0,Y 264.951,Z 557.153,A -85,B 0,C 180,E1 6829.555,E2 6829.555} C_VEL
LIN {X 0,Y 266.868,Z 561.735,A -85,B 0,C 180,E1 6827.012,E2 6827.012} C_VEL
LIN {X 0,Y 258.228,Z 641.154,A -85,B 0,C 180,E1 6825.514,E2 6825.514} C_VEL
LIN {X 0,Y 253.879,Z 663.791,A -85,B 0,C 180,E1 6824.955,E2 6824.955} C_VEL
LIN {X 0,Y 249.146,Z 681.162,A -85,B 0,C 180,E1 6824.392,E2 6824.392} C_VEL
LIN {X 0,Y 243.109,Z 698.901,A -85,B 0,C 180,E1 6823.63,E2 6823.63} C_VEL
LIN {X 0,Y 234.831,Z 718.413,A -85,B 0,C 180,E1 6822.499,E2 6822.499} C_VEL
LIN {X 0,Y 226.93,Z 734.065,A -85,B 0,C 180,E1 6821.31,E2 6821.31} C_VEL
LIN {X 0,Y 217.868,Z 749.717,A -85,B 0,C 180,E1 6819.798,E2 6819.798} C_VEL
LIN {X 0,Y 206.059,Z 767.223,A -85,B 0,C 180,E1 6817.568,E2 6817.568} C_VEL
LIN {X 0,Y 196.231,Z 780.043,A -85,B 0,C 180,E1 6815.435,E2 6815.435} C_VEL
LIN {X 0,Y 185.343,Z 792.888,A -85,B 0,C 180,E1 6812.694,E2 6812.694} C_VEL
LIN {X 0,Y 172.068,Z 806.826,A -85,B 0,C 180,E1 6808.668,E2 6808.668} C_VEL
LIN {X 0,Y 161.601,Z 816.82,A -85,B 0,C 180,E1 6804.755,E2 6804.755} C_VEL
LIN {X 0,Y 150.776,Z 826.505,A -85,B 0,C 180,E1 6799.693,E2 6799.693} C_VEL
LIN {X 0,Y 140.246,Z 835.303,A -85,B 0,C 180,E1 6793.188,E2 6793.188} C_VEL
LIN {X 0,Y 132.491,Z 841.663,A -85,B 0,C 180,E1 6786.596,E2 6786.596} C_VEL
LIN {X 0,Y 126.255,Z 847.003,A -85,B 0,C 180,E1 6778.886,E2 6778.886} C_VEL
LIN {X 0,Y 121.709,Z 851.42,A -85,B 0,C 180,E1 6769.085,E2 6769.085} C_VEL
LIN {X 0,Y 120.191,Z 853.61,A -85,B 0,C 180,E1 6760.91,E2 6760.91} C_VEL
LIN {X 0,Y 119.999,Z 854.526,A -85,B 0,C 180,E1 6754.301,E2 6754.301} C_VEL
LIN {X 0,Y 120.029,Z 854.68,A -85,B 0,C 180,E1 6748.091,E2 6748.091} C_VEL
LIN {X 0,Y 120.07,Z 853.953,A -85,B 0,C 180,E1 6740.897,E2 6740.897} C_VEL
LIN {X 0,Y 121.214,Z 851.996,A -85,B 0,C 180,E1 6732.726,E2 6732.726} C_VEL
LIN {X 0,Y 122.183,Z 850.951,A -85,B 0,C 180,E1 6729.45,E2 6729.45} C_VEL
LIN {X 0,Y 122.623,Z 849.689,A -85,B 0,C 180,E1 6725.868,E2 6725.868} C_VEL
LIN {X 0,Y 121.89,Z 846.048,A -85,B 0,C 180,E1 6717.906,E2 6717.906} C_VEL
LIN {X 0,Y 123.346,Z 843.578,A -85,B 0,C 180,E1 6713.957,E2 6713.957} C_VEL
LIN {X 0,Y 123.92,Z 843.063,A -85,B 0,C 180,E1 6713.269,E2 6713.269} C_VEL
LIN {X 0,Y 132.245,Z 836.671,A -85,B 0,C 180,E1 6705.928,E2 6705.928} C_VEL
LIN {X 0,Y 141.348,Z 829.606,A -85,B 0,C 180,E1 6700.088,E2 6700.088} C_VEL
LIN {X 0,Y 153.538,Z 819.684,A -85,B 0,C 180,E1 6694.207,E2 6694.207} C_VEL
LIN {X 0,Y 165.741,Z 808.664,A -85,B 0,C 180,E1 6689.663,E2 6689.663} C_VEL
LIN {X 0,Y 176.415,Z 798.203,A -85,B 0,C 180,E1 6686.432,E2 6686.432} C_VEL
LIN {X 0,Y 189.269,Z 784.307,A -85,B 0,C 180,E1 6683.195,E2 6683.195} C_VEL
LIN {X 0,Y 200.967,Z 769.789,A -85,B 0,C 180,E1 6680.721,E2 6680.721} C_VEL
LIN {X 0,Y 210.84,Z 756.059,A -85,B 0,C 180,E1 6678.906,E2 6678.906} C_VEL
LIN {X 0,Y 221.809,Z 738.667,A -85,B 0,C 180,E1 6677.135,E2 6677.135} C_VEL
LIN {X 0,Y 230.729,Z 721.858,A -85,B 0,C 180,E1 6675.846,E2 6675.846} C_VEL
LIN {X 0,Y 237.96,Z 706.009,A -85,B 0,C 180,E1 6674.899,E2 6674.899} C_VEL
LIN {X 0,Y 245.268,Z 686.869,A -85,B 0,C 180,E1 6674.023,E2 6674.023} C_VEL
LIN {X 0,Y 251.015,Z 667.121,A -85,B 0,C 180,E1 6673.379,E2 6673.379} C_VEL
LIN {X 0,Y 254.882,Z 649.527,A -85,B 0,C 180,E1 6672.936,E2 6672.936} C_VEL
LIN {X 0,Y 258.28,Z 625.414,A -85,B 0,C 180,E1 6672.45,E2 6672.45} C_VEL
LIN {X 0,Y 264.532,Z 567.009,A -85,B 0,C 180,E1 6671.344,E2 6671.344} C_VEL
LIN {X 0,Y 262.816,Z 562.887,A -85,B 0,C 180,E1 6668.652,E2 6668.652} C_VEL
LIN {X 0,Y 261.638,Z 560.055,A -85,B 0,C 180,E1 6666.152,E2 6666.152} C_VEL
LIN {X 0,Y 260.555,Z 556.321,A -85,B 0,C 180,E1 6661.109,E2 6661.109} C_VEL
LIN {X 0,Y 260.587,Z 556.509,A -85,B 0,C 180,E1 6658.031,E2 6658.031} C_VEL
LIN {X 0,Y 262.014,Z 560.88,A -85,B 0,C 180,E1 6652.555,E2 6652.555} C_VEL
LIN {X 0,Y 263.583,Z 564.778,A -85,B 0,C 180,E1 6649.63,E2 6649.63} C_VEL
LIN {X 0,Y 265.599,Z 569.666,A -85,B 0,C 180,E1 6646.846,E2 6646.846} C_VEL
LIN {X 0,Y 272.98,Z 583.196,A -85,B 0,C 180,E1 6640.207,E2 6640.207} C_VEL
LIN {X 0,Y 282.252,Z 593.365,A -85,B 0,C 180,E1 6634.855,E2 6634.855} C_VEL
LIN {X 0,Y 294.458,Z 602.889,A -85,B 0,C 180,E1 6629.618,E2 6629.618} C_VEL
LIN {X 0,Y 301.813,Z 608.659,A -85,B 0,C 180,E1 6626.423,E2 6626.423} C_VEL
LIN {X 0,Y 308.057,Z 613.402,A -85,B 0,C 180,E1 6623.459,E2 6623.459} C_VEL
LIN {X 0,Y 313.326,Z 618.01,A -85,B 0,C 180,E1 6620.591,E2 6620.591} C_VEL
LIN {X 0,Y 317.389,Z 621.389,A -85,B 0,C 180,E1 6618.234,E2 6618.234} C_VEL
LIN {X 0,Y 322.707,Z 626.167,A -85,B 0,C 180,E1 6614.943,E2 6614.943} C_VEL
LIN {X 0,Y 326.604,Z 629.322,A -85,B 0,C 180,E1 6612.472,E2 6612.472} C_VEL
LIN {X 0,Y 331.771,Z 634.015,A -85,B 0,C 180,E1 6608.982,E2 6608.982} C_VEL
LIN {X 0,Y 335.871,Z 637.089,A -85,B 0,C 180,E1 6606.115,E2 6606.115} C_VEL
LIN {X 0,Y 340.195,Z 641.158,A -85,B 0,C 180,E1 6602.819,E2 6602.819} C_VEL
LIN {X 0,Y 344.383,Z 644.144,A -85,B 0,C 180,E1 6599.447,E2 6599.447} C_VEL
LIN {X 0,Y 346.171,Z 645.498,A -85,B 0,C 180,E1 6597.898,E2 6597.898} C_VEL
LIN {X 0,Y 349.611,Z 648.945,A -85,B 0,C 180,E1 6594.596,E2 6594.596} C_VEL
LIN {X 0,Y 352.826,Z 651.369,A -85,B 0,C 180,E1 6591.228,E2 6591.228} C_VEL
LIN {X 0,Y 355.701,Z 652.892,A -85,B 0,C 180,E1 6587.841,E2 6587.841} C_VEL
LIN {X 0,Y 357.091,Z 653.808,A -85,B 0,C 180,E1 6585.926,E2 6585.926} C_VEL
LIN {X 0,Y 358.833,Z 656.087,A -85,B 0,C 180,E1 6582.825,E2 6582.825} C_VEL
LIN {X 0,Y 360.422,Z 657.675,A -85,B 0,C 180,E1 6579.42,E2 6579.42} C_VEL
LIN {X 0,Y 361.554,Z 658.573,A -85,B 0,C 180,E1 6576.191,E2 6576.191} C_VEL
LIN {X 0,Y 362.157,Z 659.05,A -85,B 0,C 180,E1 6572.848,E2 6572.848} C_VEL
LIN {X 0,Y 362.33,Z 659.173,A -85,B 0,C 180,E1 6569.368,E2 6569.368} C_VEL
LIN {X 0,Y 362.045,Z 658.946,A -85,B 0,C 180,E1 6566.041,E2 6566.041} C_VEL
LIN {X 0,Y 361.165,Z 658.33,A -85,B 0,C 180,E1 6562.684,E2 6562.684} C_VEL
LIN {X 0,Y 359.866,Z 657.181,A -85,B 0,C 180,E1 6559.272,E2 6559.272} C_VEL
LIN {X 0,Y 358.214,Z 655.315,A -85,B 0,C 180,E1 6555.946,E2 6555.946} C_VEL
LIN {X 0,Y 356.322,Z 653.144,A -85,B 0,C 180,E1 6553.033,E2 6553.033} C_VEL
LIN {X 0,Y 353.582,Z 651.844,A -85,B 0,C 180,E1 6549.647,E2 6549.647} C_VEL
LIN {X 0,Y 350.704,Z 649.824,A -85,B 0,C 180,E1 6546.476,E2 6546.476} C_VEL
LIN {X 0,Y 347.316,Z 646.702,A -85,B 0,C 180,E1 6543.13,E2 6543.13} C_VEL
LIN {X 0,Y 345.003,Z 644.479,A -85,B 0,C 180,E1 6541.05,E2 6541.05} C_VEL
LIN {X 0,Y 340.933,Z 641.741,A -85,B 0,C 180,E1 6537.742,E2 6537.742} C_VEL
LIN {X 0,Y 336.556,Z 637.806,A -85,B 0,C 180,E1 6534.39,E2 6534.39} C_VEL
LIN {X 0,Y 334.23,Z 635.768,A -85,B 0,C 180,E1 6532.708,E2 6532.708} C_VEL
LIN {X 0,Y 329.329,Z 631.95,A -85,B 0,C 180,E1 6529.361,E2 6529.361} C_VEL
LIN {X 0,Y 324.376,Z 627.394,A -85,B 0,C 180,E1 6526.091,E2 6526.091} C_VEL
LIN {X 0,Y 318.793,Z 622.78,A -85,B 0,C 180,E1 6522.631,E2 6522.631} C_VEL
LIN {X 0,Y 314.845,Z 619.147,A -85,B 0,C 180,E1 6520.246,E2 6520.246} C_VEL
LIN {X 0,Y 309.699,Z 614.93,A -85,B 0,C 180,E1 6517.422,E2 6517.422} C_VEL
LIN {X 0,Y 304.725,Z 610.74,A -85,B 0,C 180,E1 6514.905,E2 6514.905} C_VEL
LIN {X 0,Y 298.21,Z 605.827,A -85,B 0,C 180,E1 6511.976,E2 6511.976} C_VEL
LIN {X 0,Y 293.137,Z 602.018,A -85,B 0,C 180,E1 6509.855,E2 6509.855} C_VEL
LIN {X 0,Y 276.87,Z 588.031,A -85,B 0,C 180,E1 6502.272,E2 6502.272} C_VEL
LIN {X 0,Y 268.993,Z 576.916,A -85,B 0,C 180,E1 6496.676,E2 6496.676} C_VEL
LIN {X 0,Y 264.234,Z 566.271,A -85,B 0,C 180,E1 6491.338,E2 6491.338} C_VEL
LIN {X 0,Y 262.58,Z 562.386,A -85,B 0,C 180,E1 6488.64,E2 6488.64} C_VEL
LIN {X 0,Y 261.645,Z 560.02,A -85,B 0,C 180,E1 6486.573,E2 6486.573} C_VEL
LIN {X 0,Y 260.559,Z 556.293,A -85,B 0,C 180,E1 6481.53,E2 6481.53} C_VEL
LIN {X 0,Y 260.587,Z 556.503,A -85,B 0,C 180,E1 6478.451,E2 6478.451} C_VEL
LIN {X 0,Y 262.056,Z 561.025,A -85,B 0,C 180,E1 6472.868,E2 6472.868} C_VEL
LIN {X 0,Y 263.725,Z 565.038,A -85,B 0,C 180,E1 6469.837,E2 6469.837} C_VEL
LIN {X 0,Y 264.55,Z 567.299,A -85,B 0,C 180,E1 6468.599,E2 6468.599} C_VEL
LIN {X 0,Y 256.311,Z 641.123,A -85,B 0,C 180,E1 6467.247,E2 6467.247} C_VEL
LIN {X 0,Y 251.915,Z 663.554,A -85,B 0,C 180,E1 6466.718,E2 6466.718} C_VEL
LIN {X 0,Y 247.105,Z 680.924,A -85,B 0,C 180,E1 6466.187,E2 6466.187} C_VEL
LIN {X 0,Y 241.037,Z 698.465,A -85,B 0,C 180,E1 6465.476,E2 6465.476} C_VEL
LIN {X 0,Y 232.533,Z 718.174,A -85,B 0,C 180,E1 6464.395,E2 6464.395} C_VEL
LIN {X 0,Y 224.47,Z 733.826,A -85,B 0,C 180,E1 6463.265,E2 6463.265} C_VEL
LIN {X 0,Y 215.204,Z 749.476,A -85,B 0,C 180,E1 6461.823,E2 6461.823} C_VEL
LIN {X 0,Y 203.096,Z 766.982,A -85,B 0,C 180,E1 6459.688,E2 6459.688} C_VEL
LIN {X 0,Y 193.189,Z 779.558,A -85,B 0,C 180,E1 6457.679,E2 6457.679} C_VEL
LIN {X 0,Y 181.967,Z 792.395,A -85,B 0,C 180,E1 6455.04,E2 6455.04} C_VEL
LIN {X 0,Y 168.709,Z 805.88,A -85,B 0,C 180,E1 6451.295,E2 6451.295} C_VEL
LIN {X 0,Y 157.714,Z 815.956,A -85,B 0,C 180,E1 6447.475,E2 6447.475} C_VEL
LIN {X 0,Y 146.876,Z 825.174,A -85,B 0,C 180,E1 6442.793,E2 6442.793} C_VEL
LIN {X 0,Y 134.369,Z 835.06,A -85,B 0,C 180,E1 6435.588,E2 6435.588} C_VEL
LIN {X 0,Y 125.989,Z 841.42,A -85,B 0,C 180,E1 6428.824,E2 6428.824} C_VEL
LIN {X 0,Y 119.143,Z 846.76,A -85,B 0,C 180,E1 6420.791,E2 6420.791} C_VEL
LIN {X 0,Y 114.068,Z 851.149,A -85,B 0,C 180,E1 6410.525,E2 6410.525} C_VEL
LIN {X 0,Y 112.266,Z 853.348,A -85,B 0,C 180,E1 6401.82,E2 6401.82} C_VEL
LIN {X 0,Y 111.999,Z 854.289,A -85,B 0,C 180,E1 6394.608,E2 6394.608} C_VEL
LIN {X 0,Y 112.038,Z 854.473,A -85,B 0,C 180,E1 6388.466,E2 6388.466} C_VEL
LIN {X 0,Y 112.076,Z 853.805,A -85,B 0,C 180,E1 6380.76,E2 6380.76} C_VEL
LIN {X 0,Y 113.332,Z 851.907,A -85,B 0,C 180,E1 6372.015,E2 6372.015} C_VEL
LIN {X 0,Y 116.574,Z 848.838,A -85,B 0,C 180,E1 6363.513,E2 6363.513} C_VEL
LIN {X 0,Y 123.068,Z 843.75,A -85,B 0,C 180,E1 6354.201,E2 6354.201} C_VEL
LIN {X 0,Y 123.92,Z 843.063,A -85,B 0,C 180,E1 6353.269,E2 6353.269} C_VEL
LIN {X 0,Y 126.108,Z 840.714,A -85,B 0,C 180,E1 6350.029,E2 6350.029} C_VEL
LIN {X 0,Y 130.539,Z 833.995,A -85,B 0,C 180,E1 6341.237,E2 6341.237} C_VEL
LIN {X 0,Y 133.511,Z 831.368,A -85,B 0,C 180,E1 6338.911,E2 6338.911} C_VEL
LIN {X 0,Y 144.121,Z 823.298,A -85,B 0,C 180,E1 6333.644,E2 6333.644} C_VEL
LIN {X 0,Y 156.454,Z 813.229,A -85,B 0,C 180,E1 6328.895,E2 6328.895} C_VEL
LIN {X 0,Y 169.703,Z 801.135,A -85,B 0,C 180,E1 6324.864,E2 6324.864} C_VEL
LIN {X 0,Y 181.163,Z 789.478,A -85,B 0,C 180,E1 6322,E2 6322} C_VEL
LIN {X 0,Y 193.041,Z 776.059,A -85,B 0,C 180,E1 6319.5,E2 6319.5} C_VEL
LIN {X 0,Y 205.65,Z 759.668,A -85,B 0,C 180,E1 6317.234,E2 6317.234} C_VEL
LIN {X 0,Y 215.502,Z 744.967,A -85,B 0,C 180,E1 6315.698,E2 6315.698} C_VEL
LIN {X 0,Y 225.462,Z 727.942,A -85,B 0,C 180,E1 6314.314,E2 6314.314} C_VEL
LIN {X 0,Y 234.476,Z 709.319,A -85,B 0,C 180,E1 6313.189,E2 6313.189} C_VEL
LIN {X 0,Y 241.115,Z 692.935,A -85,B 0,C 180,E1 6312.434,E2 6312.434} C_VEL
LIN {X 0,Y 247.597,Z 673.409,A -85,B 0,C 180,E1 6311.758,E2 6311.758} C_VEL
LIN {X 0,Y 252.465,Z 653.065,A -85,B 0,C 180,E1 6311.25,E2 6311.25} C_VEL
LIN {X 0,Y 255.413,Z 635.335,A -85,B 0,C 180,E1 6310.887,E2 6310.887} C_VEL
LIN {X 0,Y 262.439,Z 572.749,A -85,B 0,C 180,E1 6309.77,E2 6309.77} C_VEL
LIN {X 0,Y 261.052,Z 569.27,A -85,B 0,C 180,E1 6307.16,E2 6307.16} C_VEL
LIN {X 0,Y 260.479,Z 567.793,A -85,B 0,C 180,E1 6305.737,E2 6305.737} C_VEL
LIN {X 0,Y 259.561,Z 564.252,A -85,B 0,C 180,E1 6300.892,E2 6300.892} C_VEL
LIN {X 0,Y 259.589,Z 564.406,A -85,B 0,C 180,E1 6298.244,E2 6298.244} C_VEL
LIN {X 0,Y 260.875,Z 568.715,A -85,B 0,C 180,E1 6292.855,E2 6292.855} C_VEL
LIN {X 0,Y 262.305,Z 572.494,A -85,B 0,C 180,E1 6290.023,E2 6290.023} C_VEL
LIN {X 0,Y 264.139,Z 577.273,A -85,B 0,C 180,E1 6287.328,E2 6287.328} C_VEL
LIN {X 0,Y 271.277,Z 590.746,A -85,B 0,C 180,E1 6280.638,E2 6280.638} C_VEL
LIN {X 0,Y 280.366,Z 600.909,A -85,B 0,C 180,E1 6275.238,E2 6275.238} C_VEL
LIN {X 0,Y 292.682,Z 610.587,A -85,B 0,C 180,E1 6269.868,E2 6269.868} C_VEL
LIN {X 0,Y 300.156,Z 616.385,A -85,B 0,C 180,E1 6266.671,E2 6266.671} C_VEL
LIN {X 0,Y 306.076,Z 620.827,A -85,B 0,C 180,E1 6263.882,E2 6263.882} C_VEL
LIN {X 0,Y 312.018,Z 625.883,A -85,B 0,C 180,E1 6260.75,E2 6260.75} C_VEL
LIN {X 0,Y 315.925,Z 629.148,A -85,B 0,C 180,E1 6258.482,E2 6258.482} C_VEL
LIN {X 0,Y 321.436,Z 634.033,A -85,B 0,C 180,E1 6255.096,E2 6255.096} C_VEL
LIN {X 0,Y 325.186,Z 637.073,A -85,B 0,C 180,E1 6252.72,E2 6252.72} C_VEL
LIN {X 0,Y 330.243,Z 641.653,A -85,B 0,C 180,E1 6249.328,E2 6249.328} C_VEL
LIN {X 0,Y 334.668,Z 645.006,A -85,B 0,C 180,E1 6246.248,E2 6246.248} C_VEL
LIN {X 0,Y 338.987,Z 649.017,A -85,B 0,C 180,E1 6242.973,E2 6242.973} C_VEL
LIN {X 0,Y 343.081,Z 651.937,A -85,B 0,C 180,E1 6239.698,E2 6239.698} C_VEL
LIN {X 0,Y 344.967,Z 653.332,A -85,B 0,C 180,E1 6238.082,E2 6238.082} C_VEL
LIN {X 0,Y 348.454,Z 656.793,A -85,B 0,C 180,E1 6234.766,E2 6234.766} C_VEL
LIN {X 0,Y 351.597,Z 659.16,A -85,B 0,C 180,E1 6231.521,E2 6231.521} C_VEL
LIN {X 0,Y 354.523,Z 660.755,A -85,B 0,C 180,E1 6228.073,E2 6228.073} C_VEL
LIN {X 0,Y 355.948,Z 661.617,A -85,B 0,C 180,E1 6226.146,E2 6226.146} C_VEL
LIN {X 0,Y 357.797,Z 663.999,A -85,B 0,C 180,E1 6222.918,E2 6222.918} C_VEL
LIN {X 0,Y 359.434,Z 665.614,A -85,B 0,C 180,E1 6219.446,E2 6219.446} C_VEL
LIN {X 0,Y 360.569,Z 666.513,A -85,B 0,C 180,E1 6216.208,E2 6216.208} C_VEL
LIN {X 0,Y 361.178,Z 666.99,A -85,B 0,C 180,E1 6212.856,E2 6212.856} C_VEL
LIN {X 0,Y 361.354,Z 667.114,A -85,B 0,C 180,E1 6209.366,E2 6209.366} C_VEL
LIN {X 0,Y 361.069,Z 666.886,A -85,B 0,C 180,E1 6206.03,E2 6206.03} C_VEL
LIN {X 0,Y 360.182,Z 666.268,A -85,B 0,C 180,E1 6202.664,E2 6202.664} C_VEL
LIN {X 0,Y 358.869,Z 665.122,A -85,B 0,C 180,E1 6199.242,E2 6199.242} C_VEL
LIN {X 0,Y 357.202,Z 663.265,A -85,B 0,C 180,E1 6195.906,E2 6195.906} C_VEL
LIN {X 0,Y 355.301,Z 661.073,A -85,B 0,C 180,E1 6192.983,E2 6192.983} C_VEL
LIN {X 0,Y 352.384,Z 659.68,A -85,B 0,C 180,E1 6189.416,E2 6189.416} C_VEL
LIN {X 0,Y 349.216,Z 657.439,A -85,B 0,C 180,E1 6186.011,E2 6186.011} C_VEL
LIN {X 0,Y 345.858,Z 654.288,A -85,B 0,C 180,E1 6182.731,E2 6182.731} C_VEL
LIN {X 0,Y 343.874,Z 652.377,A -85,B 0,C 180,E1 6180.951,E2 6180.951} C_VEL
LIN {X 0,Y 339.914,Z 649.747,A -85,B 0,C 180,E1 6177.738,E2 6177.738} C_VEL
LIN {X 0,Y 335.563,Z 645.93,A -85,B 0,C 180,E1 6174.415,E2 6174.415} C_VEL
LIN {X 0,Y 333.153,Z 643.726,A -85,B 0,C 180,E1 6172.668,E2 6172.668} C_VEL
LIN {X 0,Y 328.232,Z 639.967,A -85,B 0,C 180,E1 6169.316,E2 6169.316} C_VEL
LIN {X 0,Y 322.938,Z 635.143,A -85,B 0,C 180,E1 6165.844,E2 6165.844} C_VEL
LIN {X 0,Y 317.508,Z 630.695,A -85,B 0,C 180,E1 6162.489,E2 6162.489} C_VEL
LIN {X 0,Y 313.2,Z 626.768,A -85,B 0,C 180,E1 6159.903,E2 6159.903} C_VEL
LIN {X 0,Y 307.71,Z 622.279,A -85,B 0,C 180,E1 6156.935,E2 6156.935} C_VEL
LIN {X 0,Y 302.721,Z 618.211,A -85,B 0,C 180,E1 6154.49,E2 6154.49} C_VEL
LIN {X 0,Y 296.289,Z 613.394,A -85,B 0,C 180,E1 6151.639,E2 6151.639} C_VEL
LIN {X 0,Y 290.722,Z 609.271,A -85,B 0,C 180,E1 6149.334,E2 6149.334} C_VEL
LIN {X 0,Y 274.917,Z 595.393,A -85,B 0,C 180,E1 6141.764,E2 6141.764} C_VEL
LIN {X 0,Y 267.233,Z 584.173,A -85,B 0,C 180,E1 6136.063,E2 6136.063} C_VEL
LIN {X 0,Y 262.781,Z 573.656,A -85,B 0,C 180,E1 6130.735,E2 6130.735} C_VEL
LIN {X 0,Y 261.307,Z 569.944,A -85,B 0,C 180,E1 6128.129,E2 6128.129} C_VEL
LIN {X 0,Y 260.487,Z 567.757,A -85,B 0,C 180,E1 6126.16,E2 6126.16} C_VEL
LIN {X 0,Y 259.565,Z 564.224,A -85,B 0,C 180,E1 6121.315,E2 6121.315} C_VEL
LIN {X 0,Y 259.589,Z 564.397,A -85,B 0,C 180,E1 6118.666,E2 6118.666} C_VEL
LIN {X 0,Y 260.871,Z 568.715,A -85,B 0,C 180,E1 6113.278,E2 6113.278} C_VEL
LIN {X 0,Y 262.373,Z 572.58,A -85,B 0,C 180,E1 6110.338,E2 6110.338} C_VEL
LIN {X 0,Y 262.415,Z 573.073,A -85,B 0,C 180,E1 6110.209,E2 6110.209} C_VEL
LIN {X 0,Y 254.631,Z 641.093,A -85,B 0,C 180,E1 6109.005,E2 6109.005} C_VEL
LIN {X 0,Y 250.164,Z 663.431,A -85,B 0,C 180,E1 6108.504,E2 6108.504} C_VEL
LIN {X 0,Y 245.312,Z 680.687,A -85,B 0,C 180,E1 6108.009,E2 6108.009} C_VEL
LIN {X 0,Y 239.262,Z 697.913,A -85,B 0,C 180,E1 6107.356,E2 6107.356} C_VEL
LIN {X 0,Y 230.493,Z 717.936,A -85,B 0,C 180,E1 6106.327,E2 6106.327} C_VEL
LIN {X 0,Y 222.276,Z 733.587,A -85,B 0,C 180,E1 6105.262,E2 6105.262} C_VEL
LIN {X 0,Y 212.807,Z 749.251,A -85,B 0,C 180,E1 6103.895,E2 6103.895} C_VEL
LIN {X 0,Y 200.858,Z 766.181,A -85,B 0,C 180,E1 6101.945,E2 6101.945} C_VEL
LIN {X 0,Y 190.037,Z 779.562,A -85,B 0,C 180,E1 6099.906,E2 6099.906} C_VEL
LIN {X 0,Y 178.673,Z 792.154,A -85,B 0,C 180,E1 6097.415,E2 6097.415} C_VEL
LIN {X 0,Y 164.349,Z 806.16,A -85,B 0,C 180,E1 6093.618,E2 6093.618} C_VEL
LIN {X 0,Y 152.719,Z 816.335,A -85,B 0,C 180,E1 6089.79,E2 6089.79} C_VEL
LIN {X 0,Y 140.706,Z 826.019,A -85,B 0,C 180,E1 6084.802,E2 6084.802} C_VEL
LIN {X 0,Y 128.249,Z 835.165,A -85,B 0,C 180,E1 6077.874,E2 6077.874} C_VEL
LIN {X 0,Y 119.223,Z 841.514,A -85,B 0,C 180,E1 6070.853,E2 6070.853} C_VEL
LIN {X 0,Y 111.154,Z 847.319,A -85,B 0,C 180,E1 6061.447,E2 6061.447} C_VEL
LIN {X 0,Y 106.103,Z 851.211,A -85,B 0,C 180,E1 6050.982,E2 6050.982} C_VEL
LIN {X 0,Y 104.264,Z 853.245,A -85,B 0,C 180,E1 6041.905,E2 6041.905} C_VEL
LIN {X 0,Y 104.003,Z 854.083,A -85,B 0,C 180,E1 6034.411,E2 6034.411} C_VEL
LIN {X 0,Y 104.038,Z 854.237,A -85,B 0,C 180,E1 6028.348,E2 6028.348} C_VEL
LIN {X 0,Y 104.113,Z 853.567,A -85,B 0,C 180,E1 6020.046,E2 6020.046} C_VEL
LIN {X 0,Y 105.617,Z 851.666,A -85,B 0,C 180,E1 6010.651,E2 6010.651} C_VEL
LIN {X 0,Y 109.309,Z 848.597,A -85,B 0,C 180,E1 6001.599,E2 6001.599} C_VEL
LIN {X 0,Y 116.507,Z 843.507,A -85,B 0,C 180,E1 5991.838,E2 5991.838} C_VEL
LIN {X 0,Y 126.468,Z 836.428,A -85,B 0,C 180,E1 5983.337,E2 5983.337} C_VEL
LIN {X 0,Y 133.511,Z 831.368,A -85,B 0,C 180,E1 5978.911,E2 5978.911} C_VEL
LIN {X 0,Y 137.097,Z 828.255,A -85,B 0,C 180,E1 5976.322,E2 5976.322} C_VEL
LIN {X 0,Y 145.089,Z 819.407,A -85,B 0,C 180,E1 5969.181,E2 5969.181} C_VEL
LIN {X 0,Y 148.825,Z 816.041,A -85,B 0,C 180,E1 5967.457,E2 5967.457} C_VEL
LIN {X 0,Y 160.668,Z 806.1,A -85,B 0,C 180,E1 5963.826,E2 5963.826} C_VEL
LIN {X 0,Y 174.847,Z 792.805,A -85,B 0,C 180,E1 5960.315,E2 5960.315} C_VEL
LIN {X 0,Y 186.956,Z 779.822,A -85,B 0,C 180,E1 5957.837,E2 5957.837} C_VEL
LIN {X 0,Y 197.593,Z 767.063,A -85,B 0,C 180,E1 5955.97,E2 5955.97} C_VEL
LIN {X 0,Y 209.801,Z 750.422,A -85,B 0,C 180,E1 5954.116,E2 5954.116} C_VEL
LIN {X 0,Y 219.897,Z 734.155,A -85,B 0,C 180,E1 5952.764,E2 5952.764} C_VEL
LIN {X 0,Y 227.788,Z 719.539,A -85,B 0,C 180,E1 5951.815,E2 5951.815} C_VEL
LIN {X 0,Y 236.221,Z 701.283,A -85,B 0,C 180,E1 5950.899,E2 5950.899} C_VEL
LIN {X 0,Y 243.323,Z 681.852,A -85,B 0,C 180,E1 5950.187,E2 5950.187} C_VEL
LIN {X 0,Y 248.347,Z 664.509,A -85,B 0,C 180,E1 5949.715,E2 5949.715} C_VEL
LIN {X 0,Y 252.793,Z 643.791,A -85,B 0,C 180,E1 5949.267,E2 5949.267} C_VEL
LIN {X 0,Y 257.346,Z 606.741,A -85,B 0,C 180,E1 5948.622,E2 5948.622} C_VEL
LIN {X 0,Y 260.5,Z 578.569,A -85,B 0,C 180,E1 5948.118,E2 5948.118} C_VEL
LIN {X 0,Y 259.414,Z 575.672,A -85,B 0,C 180,E1 5945.539,E2 5945.539} C_VEL
LIN {X 0,Y 258.57,Z 572.182,A -85,B 0,C 180,E1 5940.674,E2 5940.674} C_VEL
LIN {X 0,Y 258.594,Z 572.302,A -85,B 0,C 180,E1 5938.459,E2 5938.459} C_VEL
LIN {X 0,Y 259.703,Z 576.406,A -85,B 0,C 180,E1 5933.267,E2 5933.267} C_VEL
LIN {X 0,Y 261.039,Z 580.208,A -85,B 0,C 180,E1 5930.419,E2 5930.419} C_VEL
LIN {X 0,Y 262.814,Z 585.217,A -85,B 0,C 180,E1 5927.654,E2 5927.654} C_VEL
LIN {X 0,Y 269.59,Z 598.296,A -85,B 0,C 180,E1 5921.075,E2 5921.075} C_VEL
LIN {X 0,Y 278.492,Z 608.453,A -85,B 0,C 180,E1 5915.626,E2 5915.626} C_VEL
LIN {X 0,Y 291.13,Z 618.427,A -85,B 0,C 180,E1 5910.032,E2 5910.032} C_VEL
LIN {X 0,Y 298.309,Z 623.965,A -85,B 0,C 180,E1 5907.011,E2 5907.011} C_VEL
LIN {X 0,Y 304.48,Z 628.583,A -85,B 0,C 180,E1 5904.128,E2 5904.128} C_VEL
LIN {X 0,Y 310.304,Z 633.491,A -85,B 0,C 180,E1 5901.087,E2 5901.087} C_VEL
LIN {X 0,Y 314.441,Z 636.906,A -85,B 0,C 180,E1 5898.729,E2 5898.729} C_VEL
LIN {X 0,Y 319.776,Z 641.62,A -85,B 0,C 180,E1 5895.469,E2 5895.469} C_VEL
LIN {X 0,Y 323.752,Z 644.824,A -85,B 0,C 180,E1 5892.967,E2 5892.967} C_VEL
LIN {X 0,Y 328.846,Z 649.386,A -85,B 0,C 180,E1 5889.594,E2 5889.594} C_VEL
LIN {X 0,Y 333.412,Z 652.86,A -85,B 0,C 180,E1 5886.424,E2 5886.424} C_VEL
LIN {X 0,Y 337.786,Z 656.88,A -85,B 0,C 180,E1 5883.123,E2 5883.123} C_VEL
LIN {X 0,Y 342.004,Z 659.862,A -85,B 0,C 180,E1 5879.762,E2 5879.762} C_VEL
LIN {X 0,Y 343.799,Z 661.205,A -85,B 0,C 180,E1 5878.235,E2 5878.235} C_VEL
LIN {X 0,Y 347.292,Z 664.633,A -85,B 0,C 180,E1 5874.947,E2 5874.947} C_VEL
LIN {X 0,Y 350.547,Z 667.083,A -85,B 0,C 180,E1 5871.588,E2 5871.588} C_VEL
LIN {X 0,Y 353.485,Z 668.68,A -85,B 0,C 180,E1 5868.128,E2 5868.128} C_VEL
LIN {X 0,Y 354.933,Z 669.592,A -85,B 0,C 180,E1 5866.175,E2 5866.175} C_VEL
LIN {X 0,Y 356.793,Z 671.941,A -85,B 0,C 180,E1 5862.955,E2 5862.955} C_VEL
LIN {X 0,Y 358.389,Z 673.504,A -85,B 0,C 180,E1 5859.636,E2 5859.636} C_VEL
LIN {X 0,Y 359.522,Z 674.412,A -85,B 0,C 180,E1 5856.387,E2 5856.387} C_VEL
LIN {X 0,Y 360.158,Z 674.891,A -85,B 0,C 180,E1 5853.183,E2 5853.183} C_VEL
LIN {X 0,Y 360.428,Z 675.088,A -85,B 0,C 180,E1 5849.841,E2 5849.841} C_VEL
LIN {X 0,Y 360.125,Z 674.865,A -85,B 0,C 180,E1 5846.498,E2 5846.498} C_VEL
LIN {X 0,Y 359.349,Z 674.304,A -85,B 0,C 180,E1 5843.129,E2 5843.129} C_VEL
LIN {X 0,Y 358.219,Z 673.341,A -85,B 0,C 180,E1 5839.872,E2 5839.872} C_VEL
LIN {X 0,Y 356.531,Z 671.651,A -85,B 0,C 180,E1 5836.54,E2 5836.54} C_VEL
LIN {X 0,Y 354.409,Z 669.047,A -85,B 0,C 180,E1 5833.108,E2 5833.108} C_VEL
LIN {X 0,Y 351.654,Z 667.779,A -85,B 0,C 180,E1 5829.704,E2 5829.704} C_VEL
LIN {X 0,Y 348.751,Z 665.81,A -85,B 0,C 180,E1 5826.516,E2 5826.516} C_VEL
LIN {X 0,Y 345.267,Z 662.725,A -85,B 0,C 180,E1 5823.094,E2 5823.094} C_VEL
LIN {X 0,Y 342.608,Z 660.201,A -85,B 0,C 180,E1 5820.739,E2 5820.739} C_VEL
LIN {X 0,Y 338.568,Z 657.506,A -85,B 0,C 180,E1 5817.489,E2 5817.489} C_VEL
LIN {X 0,Y 334.084,Z 653.566,A -85,B 0,C 180,E1 5814.085,E2 5814.085} C_VEL
LIN {X 0,Y 331.46,Z 651.284,A -85,B 0,C 180,E1 5812.199,E2 5812.199} C_VEL
LIN {X 0,Y 326.539,Z 647.438,A -85,B 0,C 180,E1 5808.856,E2 5808.856} C_VEL
LIN {X 0,Y 321.492,Z 642.888,A -85,B 0,C 180,E1 5805.594,E2 5805.594} C_VEL
LIN {X 0,Y 316.059,Z 638.457,A -85,B 0,C 180,E1 5802.248,E2 5802.248} C_VEL
LIN {X 0,Y 311.635,Z 634.487,A -85,B 0,C 180,E1 5799.646,E2 5799.646} C_VEL
LIN {X 0,Y 305.942,Z 629.874,A -85,B 0,C 180,E1 5796.602,E2 5796.602} C_VEL
LIN {X 0,Y 301.251,Z 626.066,A -85,B 0,C 180,E1 5794.336,E2 5794.336} C_VEL
LIN {X 0,Y 294.981,Z 621.462,A -85,B 0,C 180,E1 5791.568,E2 5791.568} C_VEL
LIN {X 0,Y 288.725,Z 616.819,A -85,B 0,C 180,E1 5788.989,E2 5788.989} C_VEL
LIN {X 0,Y 272.987,Z 602.756,A -85,B 0,C 180,E1 5781.249,E2 5781.249} C_VEL
LIN {X 0,Y 265.505,Z 591.431,A -85,B 0,C 180,E1 5775.441,E2 5775.441} C_VEL
LIN {X 0,Y 261.357,Z 581.039,A -85,B 0,C 180,E1 5770.125,E2 5770.125} C_VEL
LIN {X 0,Y 260.007,Z 577.369,A -85,B 0,C 180,E1 5767.503,E2 5767.503} C_VEL
LIN {X 0,Y 259.342,Z 575.492,A -85,B 0,C 180,E1 5765.743,E2 5765.743} C_VEL
LIN {X 0,Y 258.573,Z 572.163,A -85,B 0,C 180,E1 5761.098,E2 5761.098} C_VEL
LIN {X 0,Y 258.597,Z 572.479,A -85,B 0,C 180,E1 5758.661,E2 5758.661} C_VEL
LIN {X 0,Y 259.739,Z 576.544,A -85,B 0,C 180,E1 5753.581,E2 5753.581} C_VEL
LIN {X 0,Y 260.499,Z 578.775,A -85,B 0,C 180,E1 5751.846,E2 5751.846} C_VEL
LIN {X 0,Y 253.194,Z 641.063,A -85,B 0,C 180,E1 5750.784,E2 5750.784} C_VEL
LIN {X 0,Y 248.689,Z 663.194,A -85,B 0,C 180,E1 5750.317,E2 5750.317} C_VEL
LIN {X 0,Y 243.769,Z 680.449,A -85,B 0,C 180,E1 5749.856,E2 5749.856} C_VEL
LIN {X 0,Y 237.63,Z 697.675,A -85,B 0,C 180,E1 5749.25,E2 5749.25} C_VEL
LIN {X 0,Y 228.721,Z 717.698,A -85,B 0,C 180,E1 5748.291,E2 5748.291} C_VEL
LIN {X 0,Y 220.358,Z 733.349,A -85,B 0,C 180,E1 5747.295,E2 5747.295} C_VEL
LIN {X 0,Y 210.71,Z 748.999,A -85,B 0,C 180,E1 5746.015,E2 5746.015} C_VEL
LIN {X 0,Y 198.489,Z 765.941,A -85,B 0,C 180,E1 5744.176,E2 5744.176} C_VEL
LIN {X 0,Y 187.794,Z 778.866,A -85,B 0,C 180,E1 5742.321,E2 5742.321} C_VEL
LIN {X 0,Y 176.552,Z 791.021,A -85,B 0,C 180,E1 5740.064,E2 5740.064} C_VEL
LIN {X 0,Y 162.304,Z 804.692,A -85,B 0,C 180,E1 5736.617,E2 5736.617} C_VEL
LIN {X 0,Y 149.534,Z 815.471,A -85,B 0,C 180,E1 5732.783,E2 5732.783} C_VEL
LIN {X 0,Y 137.565,Z 824.688,A -85,B 0,C 180,E1 5728.251,E2 5728.251} C_VEL
LIN {X 0,Y 123.424,Z 834.574,A -85,B 0,C 180,E1 5721.048,E2 5721.048} C_VEL
LIN {X 0,Y 113.655,Z 840.935,A -85,B 0,C 180,E1 5714.025,E2 5714.025} C_VEL
LIN {X 0,Y 105.258,Z 846.368,A -85,B 0,C 180,E1 5705.187,E2 5705.187} C_VEL
LIN {X 0,Y 98.952,Z 850.667,A -85,B 0,C 180,E1 5693.839,E2 5693.839} C_VEL
LIN {X 0,Y 96.459,Z 852.869,A -85,B 0,C 180,E1 5683.792,E2 5683.792} C_VEL
LIN {X 0,Y 96.001,Z 853.814,A -85,B 0,C 180,E1 5675.378,E2 5675.378} C_VEL
LIN {X 0,Y 96.038,Z 854,A -85,B 0,C 180,E1 5668.21,E2 5668.21} C_VEL
LIN {X 0,Y 96.163,Z 853.328,A -85,B 0,C 180,E1 5659.213,E2 5659.213} C_VEL
LIN {X 0,Y 97.967,Z 851.425,A -85,B 0,C 180,E1 5649.072,E2 5649.072} C_VEL
LIN {X 0,Y 102.181,Z 848.355,A -85,B 0,C 180,E1 5639.415,E2 5639.415} C_VEL
LIN {X 0,Y 110.165,Z 843.264,A -85,B 0,C 180,E1 5629.198,E2 5629.198} C_VEL
LIN {X 0,Y 120.973,Z 836.185,A -85,B 0,C 180,E1 5620.503,E2 5620.503} C_VEL
LIN {X 0,Y 131.258,Z 829.195,A -85,B 0,C 180,E1 5614.647,E2 5614.647} C_VEL
LIN {X 0,Y 144.567,Z 819.505,A -85,B 0,C 180,E1 5608.973,E2 5608.973} C_VEL
LIN {X 0,Y 148.825,Z 816.041,A -85,B 0,C 180,E1 5607.457,E2 5607.457} C_VEL
LIN {X 0,Y 153.203,Z 812.179,A -85,B 0,C 180,E1 5605.542,E2 5605.542} C_VEL
LIN {X 0,Y 162.601,Z 801.855,A -85,B 0,C 180,E1 5600.278,E2 5600.278} C_VEL
LIN {X 0,Y 167.244,Z 797.207,A -85,B 0,C 180,E1 5598.808,E2 5598.808} C_VEL
LIN {X 0,Y 181.27,Z 783.326,A -85,B 0,C 180,E1 5596.022,E2 5596.022} C_VEL
LIN {X 0,Y 193.686,Z 769.069,A -85,B 0,C 180,E1 5593.957,E2 5593.957} C_VEL
LIN {X 0,Y 204.079,Z 755.585,A -85,B 0,C 180,E1 5592.461,E2 5592.461} C_VEL
LIN {X 0,Y 215.441,Z 738.752,A -85,B 0,C 180,E1 5591.027,E2 5591.027} C_VEL
LIN {X 0,Y 225.327,Z 721.143,A -85,B 0,C 180,E1 5589.915,E2 5589.915} C_VEL
LIN {X 0,Y 232.922,Z 705.295,A -85,B 0,C 180,E1 5589.147,E2 5589.147} C_VEL
LIN {X 0,Y 240.806,Z 685.416,A -85,B 0,C 180,E1 5588.423,E2 5588.423} C_VEL
LIN {X 0,Y 246.567,Z 666.379,A -85,B 0,C 180,E1 5587.927,E2 5587.927} C_VEL
LIN {X 0,Y 250.621,Z 648.686,A -85,B 0,C 180,E1 5587.561,E2 5587.561} C_VEL
LIN {X 0,Y 254.263,Z 623.974,A -85,B 0,C 180,E1 5587.131,E2 5587.131} C_VEL
LIN {X 0,Y 258.734,Z 584.782,A -85,B 0,C 180,E1 5586.444,E2 5586.444} C_VEL
LIN {X 0,Y 258.133,Z 583.115,A -85,B 0,C 180,E1 5584.675,E2 5584.675} C_VEL
LIN {X 0,Y 257.583,Z 580.11,A -85,B 0,C 180,E1 5580.454,E2 5580.454} C_VEL
LIN {X 0,Y 257.602,Z 580.387,A -85,B 0,C 180,E1 5578.453,E2 5578.453} C_VEL
LIN {X 0,Y 258.581,Z 584.239,A -85,B 0,C 180,E1 5573.572,E2 5573.572} C_VEL
LIN {X 0,Y 259.844,Z 588.089,A -85,B 0,C 180,E1 5570.71,E2 5570.71} C_VEL
LIN {X 0,Y 261.653,Z 593.588,A -85,B 0,C 180,E1 5567.766,E2 5567.766} C_VEL
LIN {X 0,Y 268.055,Z 606.03,A -85,B 0,C 180,E1 5561.414,E2 5561.414} C_VEL
LIN {X 0,Y 276.449,Z 615.836,A -85,B 0,C 180,E1 5556.115,E2 5556.115} C_VEL
LIN {X 0,Y 289.356,Z 626.124,A -85,B 0,C 180,E1 5550.286,E2 5550.286} C_VEL
LIN {X 0,Y 296.545,Z 631.677,A -85,B 0,C 180,E1 5547.25,E2 5547.25} C_VEL
LIN {X 0,Y 302.559,Z 636.162,A -85,B 0,C 180,E1 5544.448,E2 5544.448} C_VEL
LIN {X 0,Y 308.606,Z 641.219,A -85,B 0,C 180,E1 5541.309,E2 5541.309} C_VEL
LIN {X 0,Y 312.81,Z 644.644,A -85,B 0,C 180,E1 5538.966,E2 5538.966} C_VEL
LIN {X 0,Y 318.503,Z 649.524,A -85,B 0,C 180,E1 5535.584,E2 5535.584} C_VEL
LIN {X 0,Y 322.315,Z 652.575,A -85,B 0,C 180,E1 5533.213,E2 5533.213} C_VEL
LIN {X 0,Y 327.602,Z 657.253,A -85,B 0,C 180,E1 5529.742,E2 5529.742} C_VEL
LIN {X 0,Y 332.228,Z 660.789,A -85,B 0,C 180,E1 5526.548,E2 5526.548} C_VEL
LIN {X 0,Y 336.502,Z 664.669,A -85,B 0,C 180,E1 5523.345,E2 5523.345} C_VEL
LIN {X 0,Y 340.675,Z 667.63,A -85,B 0,C 180,E1 5520.047,E2 5520.047} C_VEL
LIN {X 0,Y 342.76,Z 669.225,A -85,B 0,C 180,E1 5518.265,E2 5518.265} C_VEL
LIN {X 0,Y 346.312,Z 672.643,A -85,B 0,C 180,E1 5514.93,E2 5514.93} C_VEL
LIN {X 0,Y 349.665,Z 675.116,A -85,B 0,C 180,E1 5511.469,E2 5511.469} C_VEL
LIN {X 0,Y 352.608,Z 676.671,A -85,B 0,C 180,E1 5508.003,E2 5508.003} C_VEL
LIN {X 0,Y 353.925,Z 677.576,A -85,B 0,C 180,E1 5506.193,E2 5506.193} C_VEL
LIN {X 0,Y 355.789,Z 679.883,A -85,B 0,C 180,E1 5502.992,E2 5502.992} C_VEL
LIN {X 0,Y 357.401,Z 681.442,A -85,B 0,C 180,E1 5499.663,E2 5499.663} C_VEL
LIN {X 0,Y 358.537,Z 682.352,A -85,B 0,C 180,E1 5496.404,E2 5496.404} C_VEL
LIN {X 0,Y 359.18,Z 682.831,A -85,B 0,C 180,E1 5493.191,E2 5493.191} C_VEL
LIN {X 0,Y 359.452,Z 683.029,A -85,B 0,C 180,E1 5489.841,E2 5489.841} C_VEL
LIN {X 0,Y 359.163,Z 682.813,A -85,B 0,C 180,E1 5486.649,E2 5486.649} C_VEL
LIN {X 0,Y 358.365,Z 682.242,A -85,B 0,C 180,E1 5483.11,E2 5483.11} C_VEL
LIN {X 0,Y 357.227,Z 681.28,A -85,B 0,C 180,E1 5479.844,E2 5479.844} C_VEL
LIN {X 0,Y 355.528,Z 679.596,A -85,B 0,C 180,E1 5476.502,E2 5476.502} C_VEL
LIN {X 0,Y 353.513,Z 677.075,A -85,B 0,C 180,E1 5473.233,E2 5473.233} C_VEL
LIN {X 0,Y 350.776,Z 675.788,A -85,B 0,C 180,E1 5469.825,E2 5469.825} C_VEL
LIN {X 0,Y 347.734,Z 673.772,A -85,B 0,C 180,E1 5466.498,E2 5466.498} C_VEL
LIN {X 0,Y 344.332,Z 670.822,A -85,B 0,C 180,E1 5463.159,E2 5463.159} C_VEL
LIN {X 0,Y 341.341,Z 668.022,A -85,B 0,C 180,E1 5460.522,E2 5460.522} C_VEL
LIN {X 0,Y 337.086,Z 665.153,A -85,B 0,C 180,E1 5457.126,E2 5457.126} C_VEL
LIN {X 0,Y 332.66,Z 661.248,A -85,B 0,C 180,E1 5453.787,E2 5453.787} C_VEL
LIN {X 0,Y 329.904,Z 658.916,A -85,B 0,C 180,E1 5451.811,E2 5451.811} C_VEL
LIN {X 0,Y 324.951,Z 655.045,A -85,B 0,C 180,E1 5448.508,E2 5448.508} C_VEL
LIN {X 0,Y 320.003,Z 650.616,A -85,B 0,C 180,E1 5445.332,E2 5445.332} C_VEL
LIN {X 0,Y 314.615,Z 646.326,A -85,B 0,C 180,E1 5442.096,E2 5442.096} C_VEL
LIN {X 0,Y 309.812,Z 642.112,A -85,B 0,C 180,E1 5439.344,E2 5439.344} C_VEL
LIN {X 0,Y 303.825,Z 637.294,A -85,B 0,C 180,E1 5436.195,E2 5436.195} C_VEL
LIN {X 0,Y 299.124,Z 633.51,A -85,B 0,C 180,E1 5433.92,E2 5433.92} C_VEL
LIN {X 0,Y 292.612,Z 628.69,A -85,B 0,C 180,E1 5431.05,E2 5431.05} C_VEL
LIN {X 0,Y 284.541,Z 622.792,A -85,B 0,C 180,E1 5427.737,E2 5427.737} C_VEL
LIN {X 0,Y 270.775,Z 609.726,A -85,B 0,C 180,E1 5420.525,E2 5420.525} C_VEL
LIN {X 0,Y 263.808,Z 598.689,A -85,B 0,C 180,E1 5414.812,E2 5414.812} C_VEL
LIN {X 0,Y 260.025,Z 588.583,A -85,B 0,C 180,E1 5409.619,E2 5409.619} C_VEL
LIN {X 0,Y 258.697,Z 584.653,A -85,B 0,C 180,E1 5406.76,E2 5406.76} C_VEL
LIN {X 0,Y 258.142,Z 583.075,A -85,B 0,C 180,E1 5405.101,E2 5405.101} C_VEL
LIN {X 0,Y 257.584,Z 580.105,A -85,B 0,C 180,E1 5400.88,E2 5400.88} C_VEL
LIN {X 0,Y 257.603,Z 580.371,A -85,B 0,C 180,E1 5398.878,E2 5398.878} C_VEL
LIN {X 0,Y 258.614,Z 584.372,A -85,B 0,C 180,E1 5393.887,E2 5393.887} C_VEL
LIN {X 0,Y 258.724,Z 585.122,A -85,B 0,C 180,E1 5393.496,E2 5393.496} C_VEL
LIN {X 0,Y 252.004,Z 641.033,A -85,B 0,C 180,E1 5392.582,E2 5392.582} C_VEL
LIN {X 0,Y 247.435,Z 663.072,A -85,B 0,C 180,E1 5392.146,E2 5392.146} C_VEL
LIN {X 0,Y 242.484,Z 680.212,A -85,B 0,C 180,E1 5391.725,E2 5391.725} C_VEL
LIN {X 0,Y 236.261,Z 697.437,A -85,B 0,C 180,E1 5391.168,E2 5391.168} C_VEL
LIN {X 0,Y 227.222,Z 717.459,A -85,B 0,C 180,E1 5390.282,E2 5390.282} C_VEL
LIN {X 0,Y 218.723,Z 733.11,A -85,B 0,C 180,E1 5389.361,E2 5389.361} C_VEL
LIN {X 0,Y 208.901,Z 748.759,A -85,B 0,C 180,E1 5388.172,E2 5388.172} C_VEL
LIN {X 0,Y 196.3,Z 765.859,A -85,B 0,C 180,E1 5386.437,E2 5386.437} C_VEL
LIN {X 0,Y 184.943,Z 779.226,A -85,B 0,C 180,E1 5384.626,E2 5384.626} C_VEL
LIN {X 0,Y 172.182,Z 792.563,A -85,B 0,C 180,E1 5382.235,E2 5382.235} C_VEL
LIN {X 0,Y 157.54,Z 805.858,A -85,B 0,C 180,E1 5378.897,E2 5378.897} C_VEL
LIN {X 0,Y 145.159,Z 815.85,A -85,B 0,C 180,E1 5375.394,E2 5375.394} C_VEL
LIN {X 0,Y 131.921,Z 825.534,A -85,B 0,C 180,E1 5370.643,E2 5370.643} C_VEL
LIN {X 0,Y 118.427,Z 834.331,A -85,B 0,C 180,E1 5364.143,E2 5364.143} C_VEL
LIN {X 0,Y 107.897,Z 840.692,A -85,B 0,C 180,E1 5357.059,E2 5357.059} C_VEL
LIN {X 0,Y 98.813,Z 846.033,A -85,B 0,C 180,E1 5348.114,E2 5348.114} C_VEL
LIN {X 0,Y 91.543,Z 850.426,A -85,B 0,C 180,E1 5335.905,E2 5335.905} C_VEL
LIN {X 0,Y 88.603,Z 852.629,A -85,B 0,C 180,E1 5325.043,E2 5325.043} C_VEL
LIN {X 0,Y 88.003,Z 853.609,A -85,B 0,C 180,E1 5315.215,E2 5315.215} C_VEL
LIN {X 0,Y 88.037,Z 853.764,A -85,B 0,C 180,E1 5308.048,E2 5308.048} C_VEL
LIN {X 0,Y 88.231,Z 853.089,A -85,B 0,C 180,E1 5298.231,E2 5298.231} C_VEL
LIN {X 0,Y 90.399,Z 851.185,A -85,B 0,C 180,E1 5287.225,E2 5287.225} C_VEL
LIN {X 0,Y 95.22,Z 848.113,A -85,B 0,C 180,E1 5276.906,E2 5276.906} C_VEL
LIN {X 0,Y 104.085,Z 843.021,A -85,B 0,C 180,E1 5266.241,E2 5266.241} C_VEL
LIN {X 0,Y 115.803,Z 835.942,A -85,B 0,C 180,E1 5257.409,E2 5257.409} C_VEL
LIN {X 0,Y 126.766,Z 828.952,A -85,B 0,C 180,E1 5251.59,E2 5251.59} C_VEL
LIN {X 0,Y 140.384,Z 819.547,A -85,B 0,C 180,E1 5246.183,E2 5246.183} C_VEL
LIN {X 0,Y 154.182,Z 808.673,A -85,B 0,C 180,E1 5241.98,E2 5241.98} C_VEL
LIN {X 0,Y 166.082,Z 798.271,A -85,B 0,C 180,E1 5239.064,E2 5239.064} C_VEL
LIN {X 0,Y 167.244,Z 797.207,A -85,B 0,C 180,E1 5238.808,E2 5238.808} C_VEL
LIN {X 0,Y 171.899,Z 792.517,A -85,B 0,C 180,E1 5237.439,E2 5237.439} C_VEL
LIN {X 0,Y 181.378,Z 781.059,A -85,B 0,C 180,E1 5233.603,E2 5233.603} C_VEL
LIN {X 0,Y 185.878,Z 775.821,A -85,B 0,C 180,E1 5232.477,E2 5232.477} C_VEL
LIN {X 0,Y 186.589,Z 775.045,A -85,B 0,C 180,E1 5232.364,E2 5232.364} C_VEL
LIN {X 0,Y 199.842,Z 758.885,A -85,B 0,C 180,E1 5230.546,E2 5230.546} C_VEL
LIN {X 0,Y 210.16,Z 744.362,A -85,B 0,C 180,E1 5229.32,E2 5229.32} C_VEL
LIN {X 0,Y 220.245,Z 728.033,A -85,B 0,C 180,E1 5228.255,E2 5228.255} C_VEL
LIN {X 0,Y 229.849,Z 709.312,A -85,B 0,C 180,E1 5227.35,E2 5227.35} C_VEL
LIN {X 0,Y 236.61,Z 693.47,A -85,B 0,C 180,E1 5226.771,E2 5226.771} C_VEL
LIN {X 0,Y 242.672,Z 676.268,A -85,B 0,C 180,E1 5226.295,E2 5226.295} C_VEL
LIN {X 0,Y 248.558,Z 653.997,A -85,B 0,C 180,E1 5225.836,E2 5225.836} C_VEL
LIN {X 0,Y 251.799,Z 635.848,A -85,B 0,C 180,E1 5225.523,E2 5225.523} C_VEL
LIN {X 0,Y 257.185,Z 591.215,A -85,B 0,C 180,E1 5224.804,E2 5224.804} C_VEL
LIN {X 0,Y 256.608,Z 588.051,A -85,B 0,C 180,E1 5220.456,E2 5220.456} C_VEL
LIN {X 0,Y 256.612,Z 588.28,A -85,B 0,C 180,E1 5218.67,E2 5218.67} C_VEL
LIN {X 0,Y 257.467,Z 592.069,A -85,B 0,C 180,E1 5213.88,E2 5213.88} C_VEL
LIN {X 0,Y 258.656,Z 595.965,A -85,B 0,C 180,E1 5211.003,E2 5211.003} C_VEL
LIN {X 0,Y 266.265,Z 613.396,A -85,B 0,C 180,E1 5201.964,E2 5201.964} C_VEL
LIN {X 0,Y 274.605,Z 623.38,A -85,B 0,C 180,E1 5196.515,E2 5196.515} C_VEL
LIN {X 0,Y 287.224,Z 633.659,A -85,B 0,C 180,E1 5190.617,E2 5190.617} C_VEL
LIN {X 0,Y 294.587,Z 639.364,A -85,B 0,C 180,E1 5187.468,E2 5187.468} C_VEL
LIN {X 0,Y 300.424,Z 643.718,A -85,B 0,C 180,E1 5184.743,E2 5184.743} C_VEL
LIN {X 0,Y 306.733,Z 648.929,A -85,B 0,C 180,E1 5181.507,E2 5181.507} C_VEL
LIN {X 0,Y 311.022,Z 652.404,A -85,B 0,C 180,E1 5179.155,E2 5179.155} C_VEL
LIN {X 0,Y 316.801,Z 657.259,A -85,B 0,C 180,E1 5175.788,E2 5175.788} C_VEL
LIN {X 0,Y 320.702,Z 660.329,A -85,B 0,C 180,E1 5173.428,E2 5173.428} C_VEL
LIN {X 0,Y 326.051,Z 665,A -85,B 0,C 180,E1 5169.964,E2 5169.964} C_VEL
LIN {X 0,Y 330.62,Z 668.378,A -85,B 0,C 180,E1 5166.898,E2 5166.898} C_VEL
LIN {X 0,Y 335.219,Z 672.524,A -85,B 0,C 180,E1 5163.489,E2 5163.489} C_VEL
LIN {X 0,Y 339.383,Z 675.449,A -85,B 0,C 180,E1 5160.25,E2 5160.25} C_VEL
LIN {X 0,Y 341.454,Z 676.983,A -85,B 0,C 180,E1 5158.508,E2 5158.508} C_VEL
LIN {X 0,Y 345.001,Z 680.387,A -85,B 0,C 180,E1 5155.215,E2 5155.215} C_VEL
LIN {X 0,Y 348.477,Z 682.965,A -85,B 0,C 180,E1 5151.653,E2 5151.653} C_VEL
LIN {X 0,Y 351.411,Z 684.53,A -85,B 0,C 180,E1 5148.238,E2 5148.238} C_VEL
LIN {X 0,Y 352.86,Z 685.491,A -85,B 0,C 180,E1 5146.291,E2 5146.291} C_VEL
LIN {X 0,Y 354.785,Z 687.824,A -85,B 0,C 180,E1 5143.029,E2 5143.029} C_VEL
LIN {X 0,Y 356.414,Z 689.38,A -85,B 0,C 180,E1 5139.69,E2 5139.69} C_VEL
LIN {X 0,Y 357.492,Z 690.252,A -85,B 0,C 180,E1 5136.584,E2 5136.584} C_VEL
LIN {X 0,Y 358.202,Z 690.771,A -85,B 0,C 180,E1 5133.2,E2 5133.2} C_VEL
LIN {X 0,Y 358.491,Z 690.975,A -85,B 0,C 180,E1 5130,E2 5130} C_VEL
LIN {X 0,Y 358.185,Z 690.753,A -85,B 0,C 180,E1 5126.639,E2 5126.639} C_VEL
LIN {X 0,Y 357.41,Z 690.198,A -85,B 0,C 180,E1 5123.179,E2 5123.179} C_VEL
LIN {X 0,Y 356.31,Z 689.278,A -85,B 0,C 180,E1 5119.981,E2 5119.981} C_VEL
LIN {X 0,Y 354.609,Z 687.638,A -85,B 0,C 180,E1 5116.632,E2 5116.632} C_VEL
LIN {X 0,Y 352.608,Z 685.186,A -85,B 0,C 180,E1 5113.358,E2 5113.358} C_VEL
LIN {X 0,Y 349.961,Z 683.824,A -85,B 0,C 180,E1 5110.014,E2 5110.014} C_VEL
LIN {X 0,Y 346.957,Z 681.921,A -85,B 0,C 180,E1 5106.747,E2 5106.747} C_VEL
LIN {X 0,Y 343.447,Z 679.003,A -85,B 0,C 180,E1 5103.324,E2 5103.324} C_VEL
LIN {X 0,Y 340.168,Z 675.908,A -85,B 0,C 180,E1 5100.41,E2 5100.41} C_VEL
LIN {X 0,Y 335.918,Z 673.083,A -85,B 0,C 180,E1 5097.054,E2 5097.054} C_VEL
LIN {X 0,Y 331.371,Z 669.14,A -85,B 0,C 180,E1 5093.653,E2 5093.653} C_VEL
LIN {X 0,Y 328.583,Z 666.795,A -85,B 0,C 180,E1 5091.71,E2 5091.71} C_VEL
LIN {X 0,Y 323.22,Z 662.653,A -85,B 0,C 180,E1 5088.187,E2 5088.187} C_VEL
LIN {X 0,Y 318.163,Z 658.221,A -85,B 0,C 180,E1 5085.004,E2 5085.004} C_VEL
LIN {X 0,Y 312.348,Z 653.623,A -85,B 0,C 180,E1 5081.609,E2 5081.609} C_VEL
LIN {X 0,Y 307.784,Z 649.699,A -85,B 0,C 180,E1 5079.053,E2 5079.053} C_VEL
LIN {X 0,Y 301.528,Z 644.693,A -85,B 0,C 180,E1 5075.809,E2 5075.809} C_VEL
LIN {X 0,Y 296.776,Z 640.922,A -85,B 0,C 180,E1 5073.528,E2 5073.528} C_VEL
LIN {X 0,Y 290.026,Z 635.881,A -85,B 0,C 180,E1 5070.552,E2 5070.552} C_VEL
LIN {X 0,Y 277.196,Z 625.586,A -85,B 0,C 180,E1 5064.837,E2 5064.837} C_VEL
LIN {X 0,Y 269.193,Z 617.482,A -85,B 0,C 180,E1 5060.197,E2 5060.197} C_VEL
LIN {X 0,Y 262.19,Z 606.06,A -85,B 0,C 180,E1 5054.228,E2 5054.228} C_VEL
LIN {X 0,Y 258.656,Z 595.965,A -85,B 0,C 180,E1 5048.997,E2 5048.997} C_VEL
LIN {X 0,Y 257.467,Z 592.069,A -85,B 0,C 180,E1 5046.12,E2 5046.12} C_VEL
LIN {X 0,Y 256.609,Z 588.046,A -85,B 0,C 180,E1 5040.883,E2 5040.883} C_VEL
LIN {X 0,Y 256.613,Z 588.263,A -85,B 0,C 180,E1 5039.097,E2 5039.097} C_VEL
LIN {X 0,Y 257.169,Z 591.44,A -85,B 0,C 180,E1 5035.168,E2 5035.168} C_VEL
LIN {X 0,Y 251.004,Z 641.397,A -85,B 0,C 180,E1 5034.388,E2 5034.388} C_VEL
LIN {X 0,Y 246.406,Z 663.08,A -85,B 0,C 180,E1 5033.99,E2 5033.99} C_VEL
LIN {X 0,Y 241.458,Z 679.985,A -85,B 0,C 180,E1 5033.611,E2 5033.611} C_VEL
LIN {X 0,Y 235.16,Z 697.203,A -85,B 0,C 180,E1 5033.106,E2 5033.106} C_VEL
LIN {X 0,Y 226,Z 717.223,A -85,B 0,C 180,E1 5032.298,E2 5032.298} C_VEL
LIN {X 0,Y 217.376,Z 732.871,A -85,B 0,C 180,E1 5031.456,E2 5031.456} C_VEL
LIN {X 0,Y 207.392,Z 748.519,A -85,B 0,C 180,E1 5030.363,E2 5030.363} C_VEL
LIN {X 0,Y 194.687,Z 765.461,A -85,B 0,C 180,E1 5028.782,E2 5028.782} C_VEL
LIN {X 0,Y 183.086,Z 778.84,A -85,B 0,C 180,E1 5027.106,E2 5027.106} C_VEL
LIN {X 0,Y 170.769,Z 791.43,A -85,B 0,C 180,E1 5025.028,E2 5025.028} C_VEL
LIN {X 0,Y 155.656,Z 804.912,A -85,B 0,C 180,E1 5021.925,E2 5021.925} C_VEL
LIN {X 0,Y 142.653,Z 815.081,A -85,B 0,C 180,E1 5018.608,E2 5018.608} C_VEL
LIN {X 0,Y 129.448,Z 824.359,A -85,B 0,C 180,E1 5014.351,E2 5014.351} C_VEL
LIN {X 0,Y 113.807,Z 834.088,A -85,B 0,C 180,E1 5007.5,E2 5007.5} C_VEL
LIN {X 0,Y 102.475,Z 840.449,A -85,B 0,C 180,E1 5000.425,E2 5000.425} C_VEL
LIN {X 0,Y 92.494,Z 845.791,A -85,B 0,C 180,E1 4991.253,E2 4991.253} C_VEL
LIN {X 0,Y 84.271,Z 850.184,A -85,B 0,C 180,E1 4978.332,E2 4978.332} C_VEL
LIN {X 0,Y 80.793,Z 852.389,A -85,B 0,C 180,E1 4966.537,E2 4966.537} C_VEL
LIN {X 0,Y 80.005,Z 853.371,A -85,B 0,C 180,E1 4955.738,E2 4955.738} C_VEL
LIN {X 0,Y 80.035,Z 853.527,A -85,B 0,C 180,E1 4947.852,E2 4947.852} C_VEL
LIN {X 0,Y 80.323,Z 852.85,A -85,B 0,C 180,E1 4937.053,E2 4937.053} C_VEL
LIN {X 0,Y 83.144,Z 850.816,A -85,B 0,C 180,E1 4924.472,E2 4924.472} C_VEL
LIN {X 0,Y 88.88,Z 847.658,A -85,B 0,C 180,E1 4913.401,E2 4913.401} C_VEL
LIN {X 0,Y 98.89,Z 842.47,A -85,B 0,C 180,E1 4902.433,E2 4902.433} C_VEL
LIN {X 0,Y 111.281,Z 835.536,A -85,B 0,C 180,E1 4893.877,E2 4893.877} C_VEL
LIN {X 0,Y 123.426,Z 828.238,A -85,B 0,C 180,E1 4887.998,E2 4887.998} C_VEL
LIN {X 0,Y 138.61,Z 818.093,A -85,B 0,C 180,E1 4882.587,E2 4882.587} C_VEL
LIN {X 0,Y 152.173,Z 807.727,A -85,B 0,C 180,E1 4878.892,E2 4878.892} C_VEL
LIN {X 0,Y 164.487,Z 797.236,A -85,B 0,C 180,E1 4876.179,E2 4876.179} C_VEL
LIN {X 0,Y 178.956,Z 783.343,A -85,B 0,C 180,E1 4873.557,E2 4873.557} C_VEL
LIN {X 0,Y 186.589,Z 775.045,A -85,B 0,C 180,E1 4872.364,E2 4872.364} C_VEL
LIN {X 0,Y 191.188,Z 769.675,A -85,B 0,C 180,E1 4871.384,E2 4871.384} C_VEL
LIN {X 0,Y 201.105,Z 755.778,A -85,B 0,C 180,E1 4868.27,E2 4868.27} C_VEL
LIN {X 0,Y 205.202,Z 749.749,A -85,B 0,C 180,E1 4867.523,E2 4867.523} C_VEL
LIN {X 0,Y 215.839,Z 733.443,A -85,B 0,C 180,E1 4866.472,E2 4866.472} C_VEL
LIN {X 0,Y 224.575,Z 717.914,A -85,B 0,C 180,E1 4865.707,E2 4865.707} C_VEL
LIN {X 0,Y 233.511,Z 699.06,A -85,B 0,C 180,E1 4865.006,E2 4865.006} C_VEL
LIN {X 0,Y 240.452,Z 680.503,A -85,B 0,C 180,E1 4864.506,E2 4864.506} C_VEL
LIN {X 0,Y 245.787,Z 662.516,A -85,B 0,C 180,E1 4864.142,E2 4864.142} C_VEL
LIN {X 0,Y 250.445,Z 640.395,A -85,B 0,C 180,E1 4863.772,E2 4863.772} C_VEL
LIN {X 0,Y 255.795,Z 598.096,A -85,B 0,C 180,E1 4863.147,E2 4863.147} C_VEL
LIN {X 0,Y 255.624,Z 595.983,A -85,B 0,C 180,E1 4860.234,E2 4860.234} C_VEL
LIN {X 0,Y 255.625,Z 596.172,A -85,B 0,C 180,E1 4858.889,E2 4858.889} C_VEL
LIN {X 0,Y 256.36,Z 599.897,A -85,B 0,C 180,E1 4854.19,E2 4854.19} C_VEL
LIN {X 0,Y 257.529,Z 604.009,A -85,B 0,C 180,E1 4851.189,E2 4851.189} C_VEL
LIN {X 0,Y 264.123,Z 620.207,A -85,B 0,C 180,E1 4842.837,E2 4842.837} C_VEL
LIN {X 0,Y 272.476,Z 630.745,A -85,B 0,C 180,E1 4837.007,E2 4837.007} C_VEL
LIN {X 0,Y 284.415,Z 640.862,A -85,B 0,C 180,E1 4831.106,E2 4831.106} C_VEL
LIN {X 0,Y 292.221,Z 646.866,A -85,B 0,C 180,E1 4827.752,E2 4827.752} C_VEL
LIN {X 0,Y 298.1,Z 651.243,A -85,B 0,C 180,E1 4825.015,E2 4825.015} C_VEL
LIN {X 0,Y 304.477,Z 656.477,A -85,B 0,C 180,E1 4821.77,E2 4821.77} C_VEL
LIN {X 0,Y 308.846,Z 659.97,A -85,B 0,C 180,E1 4819.418,E2 4819.418} C_VEL
LIN {X 0,Y 314.903,Z 664.975,A -85,B 0,C 180,E1 4815.96,E2 4815.96} C_VEL
LIN {X 0,Y 318.845,Z 668.074,A -85,B 0,C 180,E1 4813.598,E2 4813.598} C_VEL
LIN {X 0,Y 324.45,Z 672.859,A -85,B 0,C 180,E1 4810.038,E2 4810.038} C_VEL
LIN {X 0,Y 328.923,Z 676.148,A -85,B 0,C 180,E1 4807.069,E2 4807.069} C_VEL
LIN {X 0,Y 333.591,Z 680.282,A -85,B 0,C 180,E1 4803.675,E2 4803.675} C_VEL
LIN {X 0,Y 338.156,Z 683.423,A -85,B 0,C 180,E1 4800.175,E2 4800.175} C_VEL
LIN {X 0,Y 340.247,Z 685.079,A -85,B 0,C 180,E1 4798.427,E2 4798.427} C_VEL
LIN {X 0,Y 344.017,Z 688.582,A -85,B 0,C 180,E1 4794.924,E2 4794.924} C_VEL
LIN {X 0,Y 347.296,Z 690.917,A -85,B 0,C 180,E1 4791.609,E2 4791.609} C_VEL
LIN {X 0,Y 350.333,Z 692.49,A -85,B 0,C 180,E1 4788.124,E2 4788.124} C_VEL
LIN {X 0,Y 351.552,Z 693.268,A -85,B 0,C 180,E1 4786.523,E2 4786.523} C_VEL
LIN {X 0,Y 353.545,Z 695.651,A -85,B 0,C 180,E1 4783.242,E2 4783.242} C_VEL
LIN {X 0,Y 355.209,Z 697.245,A -85,B 0,C 180,E1 4779.887,E2 4779.887} C_VEL
LIN {X 0,Y 356.419,Z 698.211,A -85,B 0,C 180,E1 4776.443,E2 4776.443} C_VEL
LIN {X 0,Y 357.086,Z 698.693,A -85,B 0,C 180,E1 4773.21,E2 4773.21} C_VEL
LIN {X 0,Y 357.308,Z 698.883,A -85,B 0,C 180,E1 4769.84,E2 4769.84} C_VEL
LIN {X 0,Y 357.092,Z 698.679,A -85,B 0,C 180,E1 4766.629,E2 4766.629} C_VEL
LIN {X 0,Y 356.348,Z 698.141,A -85,B 0,C 180,E1 4763.232,E2 4763.232} C_VEL
LIN {X 0,Y 355.039,Z 697.128,A -85,B 0,C 180,E1 4759.781,E2 4759.781} C_VEL
LIN {X 0,Y 353.327,Z 695.453,A -85,B 0,C 180,E1 4756.416,E2 4756.416} C_VEL
LIN {X 0,Y 351.291,Z 692.959,A -85,B 0,C 180,E1 4753.124,E2 4753.124} C_VEL
LIN {X 0,Y 348.415,Z 691.587,A -85,B 0,C 180,E1 4749.682,E2 4749.682} C_VEL
LIN {X 0,Y 345.171,Z 689.48,A -85,B 0,C 180,E1 4746.229,E2 4746.229} C_VEL
LIN {X 0,Y 341.597,Z 686.458,A -85,B 0,C 180,E1 4742.826,E2 4742.826} C_VEL
LIN {X 0,Y 338.627,Z 683.693,A -85,B 0,C 180,E1 4740.215,E2 4740.215} C_VEL
LIN {X 0,Y 334.282,Z 680.83,A -85,B 0,C 180,E1 4736.857,E2 4736.857} C_VEL
LIN {X 0,Y 329.354,Z 676.591,A -85,B 0,C 180,E1 4733.251,E2 4733.251} C_VEL
LIN {X 0,Y 326.536,Z 674.328,A -85,B 0,C 180,E1 4731.318,E2 4731.318} C_VEL
LIN {X 0,Y 321.413,Z 670.393,A -85,B 0,C 180,E1 4728.013,E2 4728.013} C_VEL
LIN {X 0,Y 316.235,Z 665.919,A -85,B 0,C 180,E1 4724.82,E2 4724.82} C_VEL
LIN {X 0,Y 310.114,Z 661.127,A -85,B 0,C 180,E1 4721.305,E2 4721.305} C_VEL
LIN {X 0,Y 305.554,Z 657.256,A -85,B 0,C 180,E1 4718.789,E2 4718.789} C_VEL
LIN {X 0,Y 299.023,Z 652.06,A -85,B 0,C 180,E1 4715.447,E2 4715.447} C_VEL
LIN {X 0,Y 294.226,Z 648.296,A -85,B 0,C 180,E1 4713.157,E2 4713.157} C_VEL
LIN {X 0,Y 287.437,Z 643.2,A -85,B 0,C 180,E1 4710.163,E2 4710.163} C_VEL
LIN {X 0,Y 275.514,Z 633.489,A -85,B 0,C 180,E1 4704.655,E2 4704.655} C_VEL
LIN {X 0,Y 267.188,Z 624.648,A -85,B 0,C 180,E1 4699.556,E2 4699.556} C_VEL
LIN {X 0,Y 260.556,Z 613.317,A -85,B 0,C 180,E1 4693.583,E2 4693.583} C_VEL
LIN {X 0,Y 257.318,Z 603.344,A -85,B 0,C 180,E1 4688.368,E2 4688.368} C_VEL
LIN {X 0,Y 256.213,Z 599.205,A -85,B 0,C 180,E1 4685.252,E2 4685.252} C_VEL
LIN {X 0,Y 255.624,Z 595.987,A -85,B 0,C 180,E1 4680.663,E2 4680.663} C_VEL
LIN {X 0,Y 255.621,Z 596.34,A -85,B 0,C 180,E1 4679.094,E2 4679.094} C_VEL
LIN {X 0,Y 255.766,Z 598.346,A -85,B 0,C 180,E1 4676.85,E2 4676.85} C_VEL
LIN {X 0,Y 250.233,Z 641.901,A -85,B 0,C 180,E1 4676.205,E2 4676.205} C_VEL
LIN {X 0,Y 245.603,Z 663.203,A -85,B 0,C 180,E1 4675.845,E2 4675.845} C_VEL
LIN {X 0,Y 240.427,Z 680.577,A -85,B 0,C 180,E1 4675.493,E2 4675.493} C_VEL
LIN {X 0,Y 233.17,Z 699.885,A -85,B 0,C 180,E1 4674.968,E2 4674.968} C_VEL
LIN {X 0,Y 224.575,Z 717.914,A -85,B 0,C 180,E1 4674.293,E2 4674.293} C_VEL
LIN {X 0,Y 215.839,Z 733.443,A -85,B 0,C 180,E1 4673.528,E2 4673.528} C_VEL
LIN {X 0,Y 204.501,Z 750.759,A -85,B 0,C 180,E1 4672.403,E2 4672.403} C_VEL
LIN {X 0,Y 192.117,Z 766.583,A -85,B 0,C 180,E1 4671.005,E2 4671.005} C_VEL
LIN {X 0,Y 180.973,Z 779.1,A -85,B 0,C 180,E1 4669.547,E2 4669.547} C_VEL
LIN {X 0,Y 166.999,Z 792.972,A -85,B 0,C 180,E1 4667.392,E2 4667.392} C_VEL
LIN {X 0,Y 152.415,Z 805.374,A -85,B 0,C 180,E1 4664.646,E2 4664.646} C_VEL
LIN {X 0,Y 139.133,Z 815.366,A -85,B 0,C 180,E1 4661.545,E2 4661.545} C_VEL
LIN {X 0,Y 124.692,Z 825.048,A -85,B 0,C 180,E1 4657.237,E2 4657.237} C_VEL
LIN {X 0,Y 109.286,Z 834.017,A -85,B 0,C 180,E1 4650.97,E2 4650.97} C_VEL
LIN {X 0,Y 97.444,Z 840.206,A -85,B 0,C 180,E1 4644.153,E2 4644.153} C_VEL
LIN {X 0,Y 86.492,Z 845.548,A -85,B 0,C 180,E1 4634.842,E2 4634.842} C_VEL
LIN {X 0,Y 77.131,Z 849.962,A -85,B 0,C 180,E1 4621.122,E2 4621.122} C_VEL
LIN {X 0,Y 72.903,Z 852.242,A -85,B 0,C 180,E1 4607.561,E2 4607.561} C_VEL
LIN {X 0,Y 72.007,Z 853.166,A -85,B 0,C 180,E1 4595.578,E2 4595.578} C_VEL
LIN {X 0,Y 72.033,Z 853.291,A -85,B 0,C 180,E1 4587.613,E2 4587.613} C_VEL
LIN {X 0,Y 72.451,Z 852.61,A -85,B 0,C 180,E1 4575.617,E2 4575.617} C_VEL
LIN {X 0,Y 75.629,Z 850.697,A -85,B 0,C 180,E1 4562.41,E2 4562.41} C_VEL
LIN {X 0,Y 81.979,Z 847.628,A -85,B 0,C 180,E1 4550.639,E2 4550.639} C_VEL
LIN {X 0,Y 92.914,Z 842.536,A -85,B 0,C 180,E1 4539.216,E2 4539.216} C_VEL
LIN {X 0,Y 106.617,Z 835.456,A -85,B 0,C 180,E1 4530.373,E2 4530.373} C_VEL
LIN {X 0,Y 118.984,Z 828.466,A -85,B 0,C 180,E1 4524.834,E2 4524.834} C_VEL
LIN {X 0,Y 133.954,Z 819.062,A -85,B 0,C 180,E1 4519.871,E2 4519.871} C_VEL
LIN {X 0,Y 148.83,Z 808.189,A -85,B 0,C 180,E1 4516.124,E2 4516.124} C_VEL
LIN {X 0,Y 161.485,Z 797.788,A -85,B 0,C 180,E1 4513.576,E2 4513.576} C_VEL
LIN {X 0,Y 175.353,Z 784.947,A -85,B 0,C 180,E1 4511.272,E2 4511.272} C_VEL
LIN {X 0,Y 189.472,Z 769.711,A -85,B 0,C 180,E1 4509.325,E2 4509.325} C_VEL
LIN {X 0,Y 200.303,Z 756.294,A -85,B 0,C 180,E1 4508.046,E2 4508.046} C_VEL
LIN {X 0,Y 205.202,Z 749.749,A -85,B 0,C 180,E1 4507.523,E2 4507.523} C_VEL
LIN {X 0,Y 209.227,Z 743.603,A -85,B 0,C 180,E1 4506.822,E2 4506.822} C_VEL
LIN {X 0,Y 218.255,Z 728.182,A -85,B 0,C 180,E1 4504.353,E2 4504.353} C_VEL
LIN {X 0,Y 221.299,Z 722.595,A -85,B 0,C 180,E1 4503.856,E2 4503.856} C_VEL
LIN {X 0,Y 221.818,Z 721.614,A -85,B 0,C 180,E1 4503.81,E2 4503.81} C_VEL
LIN {X 0,Y 229.778,Z 705.774,A -85,B 0,C 180,E1 4503.242,E2 4503.242} C_VEL
LIN {X 0,Y 237.234,Z 688.03,A -85,B 0,C 180,E1 4502.758,E2 4502.758} C_VEL
LIN {X 0,Y 244.037,Z 667.105,A -85,B 0,C 180,E1 4502.352,E2 4502.352} C_VEL
LIN {X 0,Y 248.493,Z 648.545,A -85,B 0,C 180,E1 4502.06,E2 4502.06} C_VEL
LIN {X 0,Y 252.125,Z 625.598,A -85,B 0,C 180,E1 4501.732,E2 4501.732} C_VEL
LIN {X 0,Y 254.634,Z 604.837,A -85,B 0,C 180,E1 4501.434,E2 4501.434} C_VEL
LIN {X 0,Y 254.643,Z 603.928,A -85,B 0,C 180,E1 4500.01,E2 4500.01} C_VEL
LIN {X 0,Y 254.634,Z 604.246,A -85,B 0,C 180,E1 4498.885,E2 4498.885} C_VEL
LIN {X 0,Y 255.262,Z 607.723,A -85,B 0,C 180,E1 4494.503,E2 4494.503} C_VEL
LIN {X 0,Y 256.293,Z 611.78,A -85,B 0,C 180,E1 4491.598,E2 4491.598} C_VEL
LIN {X 0,Y 262.375,Z 627.569,A -85,B 0,C 180,E1 4483.404,E2 4483.404} C_VEL
LIN {X 0,Y 270.486,Z 638.263,A -85,B 0,C 180,E1 4477.403,E2 4477.403} C_VEL
LIN {X 0,Y 282.564,Z 648.75,A -85,B 0,C 180,E1 4471.13,E2 4471.13} C_VEL
LIN {X 0,Y 290.656,Z 655.051,A -85,B 0,C 180,E1 4467.558,E2 4467.558} C_VEL
LIN {X 0,Y 296.129,Z 659.221,A -85,B 0,C 180,E1 4464.984,E2 4464.984} C_VEL
LIN {X 0,Y 302.744,Z 664.514,A -85,B 0,C 180,E1 4461.632,E2 4461.632} C_VEL
LIN {X 0,Y 307.293,Z 668.275,A -85,B 0,C 180,E1 4459.17,E2 4459.17} C_VEL
LIN {X 0,Y 313.266,Z 673.018,A -85,B 0,C 180,E1 4455.797,E2 4455.797} C_VEL
LIN {X 0,Y 317.258,Z 676.248,A -85,B 0,C 180,E1 4453.427,E2 4453.427} C_VEL
LIN {X 0,Y 322.774,Z 680.814,A -85,B 0,C 180,E1 4449.96,E2 4449.96} C_VEL
LIN {X 0,Y 326.966,Z 683.884,A -85,B 0,C 180,E1 4447.211,E2 4447.211} C_VEL
LIN {X 0,Y 331.895,Z 688.172,A -85,B 0,C 180,E1 4443.662,E2 4443.662} C_VEL
LIN {X 0,Y 336.552,Z 691.299,A -85,B 0,C 180,E1 4440.137,E2 4440.137} C_VEL
LIN {X 0,Y 338.776,Z 693.174,A -85,B 0,C 180,E1 4438.274,E2 4438.274} C_VEL
LIN {X 0,Y 342.462,Z 696.508,A -85,B 0,C 180,E1 4434.861,E2 4434.861} C_VEL
LIN {X 0,Y 345.95,Z 698.921,A -85,B 0,C 180,E1 4431.355,E2 4431.355} C_VEL
LIN {X 0,Y 348.94,Z 700.396,A -85,B 0,C 180,E1 4427.988,E2 4427.988} C_VEL
LIN {X 0,Y 350.119,Z 701.288,A -85,B 0,C 180,E1 4426.394,E2 4426.394} C_VEL
LIN {X 0,Y 352.158,Z 703.671,A -85,B 0,C 180,E1 4422.961,E2 4422.961} C_VEL
LIN {X 0,Y 353.794,Z 705.202,A -85,B 0,C 180,E1 4419.559,E2 4419.559} C_VEL
LIN {X 0,Y 354.983,Z 706.119,A -85,B 0,C 180,E1 4416.239,E2 4416.239} C_VEL
LIN {X 0,Y 355.652,Z 706.593,A -85,B 0,C 180,E1 4412.901,E2 4412.901} C_VEL
LIN {X 0,Y 355.806,Z 706.735,A -85,B 0,C 180,E1 4409.678,E2 4409.678} C_VEL
LIN {X 0,Y 355.512,Z 706.509,A -85,B 0,C 180,E1 4406.291,E2 4406.291} C_VEL
LIN {X 0,Y 354.782,Z 705.96,A -85,B 0,C 180,E1 4403.04,E2 4403.04} C_VEL
LIN {X 0,Y 353.478,Z 704.969,A -85,B 0,C 180,E1 4399.735,E2 4399.735} C_VEL
LIN {X 0,Y 351.75,Z 703.29,A -85,B 0,C 180,E1 4396.354,E2 4396.354} C_VEL
LIN {X 0,Y 349.725,Z 700.803,A -85,B 0,C 180,E1 4393.046,E2 4393.046} C_VEL
LIN {X 0,Y 347.001,Z 699.495,A -85,B 0,C 180,E1 4389.772,E2 4389.772} C_VEL
LIN {X 0,Y 343.719,Z 697.448,A -85,B 0,C 180,E1 4386.366,E2 4386.366} C_VEL
LIN {X 0,Y 340.118,Z 694.485,A -85,B 0,C 180,E1 4382.942,E2 4382.942} C_VEL
LIN {X 0,Y 336.821,Z 691.446,A -85,B 0,C 180,E1 4380.068,E2 4380.068} C_VEL
LIN {X 0,Y 332.23,Z 688.429,A -85,B 0,C 180,E1 4376.583,E2 4376.583} C_VEL
LIN {X 0,Y 327.43,Z 684.34,A -85,B 0,C 180,E1 4373.117,E2 4373.117} C_VEL
LIN {X 0,Y 324.548,Z 682.045,A -85,B 0,C 180,E1 4371.192,E2 4371.192} C_VEL
LIN {X 0,Y 319.029,Z 677.833,A -85,B 0,C 180,E1 4367.685,E2 4367.685} C_VEL
LIN {X 0,Y 314.115,Z 673.603,A -85,B 0,C 180,E1 4364.69,E2 4364.69} C_VEL
LIN {X 0,Y 307.978,Z 668.88,A -85,B 0,C 180,E1 4361.213,E2 4361.213} C_VEL
LIN {X 0,Y 303.166,Z 664.819,A -85,B 0,C 180,E1 4358.591,E2 4358.591} C_VEL
LIN {X 0,Y 296.49,Z 659.545,A -85,B 0,C 180,E1 4355.203,E2 4355.203} C_VEL
LIN {X 0,Y 291.847,Z 655.896,A -85,B 0,C 180,E1 4352.993,E2 4352.993} C_VEL
LIN {X 0,Y 284.84,Z 650.641,A -85,B 0,C 180,E1 4349.885,E2 4349.885} C_VEL
LIN {X 0,Y 267.637,Z 635.184,A -85,B 0,C 180,E1 4340.776,E2 4340.776} C_VEL
LIN {X 0,Y 259.339,Z 621.578,A -85,B 0,C 180,E1 4333.421,E2 4333.421} C_VEL
LIN {X 0,Y 256.058,Z 610.888,A -85,B 0,C 180,E1 4327.845,E2 4327.845} C_VEL
LIN {X 0,Y 255.128,Z 607.032,A -85,B 0,C 180,E1 4324.936,E2 4324.936} C_VEL
LIN {X 0,Y 254.643,Z 603.931,A -85,B 0,C 180,E1 4320.44,E2 4320.44} C_VEL
LIN {X 0,Y 254.635,Z 604.23,A -85,B 0,C 180,E1 4319.315,E2 4319.315} C_VEL
LIN {X 0,Y 254.618,Z 604.985,A -85,B 0,C 180,E1 4318.553,E2 4318.553} C_VEL
LIN {X 0,Y 249.66,Z 642.757,A -85,B 0,C 180,E1 4318.026,E2 4318.026} C_VEL
LIN {X 0,Y 244.967,Z 663.668,A -85,B 0,C 180,E1 4317.704,E2 4317.704} C_VEL
LIN {X 0,Y 239.46,Z 681.763,A -85,B 0,C 180,E1 4317.376,E2 4317.376} C_VEL
LIN {X 0,Y 231.308,Z 702.48,A -85,B 0,C 180,E1 4316.858,E2 4316.858} C_VEL
LIN {X 0,Y 222.933,Z 719.525,A -85,B 0,C 180,E1 4316.273,E2 4316.273} C_VEL
LIN {X 0,Y 213.609,Z 735.628,A -85,B 0,C 180,E1 4315.544,E2 4315.544} C_VEL
LIN {X 0,Y 200.92,Z 753.998,A -85,B 0,C 180,E1 4314.414,E2 4314.414} C_VEL
LIN {X 0,Y 189.773,Z 767.792,A -85,B 0,C 180,E1 4313.277,E2 4313.277} C_VEL
LIN {X 0,Y 176.806,Z 781.865,A -85,B 0,C 180,E1 4311.735,E2 4311.735} C_VEL
LIN {X 0,Y 161.642,Z 795.961,A -85,B 0,C 180,E1 4309.573,E2 4309.573} C_VEL
LIN {X 0,Y 148.609,Z 806.54,A -85,B 0,C 180,E1 4307.304,E2 4307.304} C_VEL
LIN {X 0,Y 134.962,Z 816.366,A -85,B 0,C 180,E1 4304.38,E2 4304.38} C_VEL
LIN {X 0,Y 117.468,Z 827.281,A -85,B 0,C 180,E1 4299.434,E2 4299.434} C_VEL
LIN {X 0,Y 103.494,Z 834.81,A -85,B 0,C 180,E1 4293.955,E2 4293.955} C_VEL
LIN {X 0,Y 90.022,Z 841.311,A -85,B 0,C 180,E1 4286.406,E2 4286.406} C_VEL
LIN {X 0,Y 76.88,Z 846.961,A -85,B 0,C 180,E1 4274.609,E2 4274.609} C_VEL
LIN {X 0,Y 69.18,Z 850.157,A -85,B 0,C 180,E1 4262.327,E2 4262.327} C_VEL
LIN {X 0,Y 64.892,Z 852.186,A -85,B 0,C 180,E1 4247.948,E2 4247.948} C_VEL
LIN {X 0,Y 64.012,Z 852.992,A -85,B 0,C 180,E1 4234.479,E2 4234.479} C_VEL
LIN {X 0,Y 64.03,Z 853.054,A -85,B 0,C 180,E1 4227.315,E2 4227.315} C_VEL
LIN {X 0,Y 64.754,Z 852.279,A -85,B 0,C 180,E1 4212.94,E2 4212.94} C_VEL
LIN {X 0,Y 68.827,Z 850.309,A -85,B 0,C 180,E1 4198.469,E2 4198.469} C_VEL
LIN {X 0,Y 76.344,Z 847.174,A -85,B 0,C 180,E1 4186.044,E2 4186.044} C_VEL
LIN {X 0,Y 89.326,Z 841.648,A -85,B 0,C 180,E1 4174.077,E2 4174.077} C_VEL
LIN {X 0,Y 102.705,Z 835.213,A -85,B 0,C 180,E1 4166.412,E2 4166.412} C_VEL
LIN {X 0,Y 115.774,Z 828.223,A -85,B 0,C 180,E1 4161.142,E2 4161.142} C_VEL
LIN {X 0,Y 131.392,Z 818.819,A -85,B 0,C 180,E1 4156.505,E2 4156.505} C_VEL
LIN {X 0,Y 147.191,Z 807.623,A -85,B 0,C 180,E1 4152.97,E2 4152.97} C_VEL
LIN {X 0,Y 159.765,Z 797.547,A -85,B 0,C 180,E1 4150.727,E2 4150.727} C_VEL
LIN {X 0,Y 173.944,Z 784.708,A -85,B 0,C 180,E1 4148.64,E2 4148.64} C_VEL
LIN {X 0,Y 188.326,Z 769.475,A -85,B 0,C 180,E1 4146.884,E2 4146.884} C_VEL
LIN {X 0,Y 199.461,Z 755.89,A -85,B 0,C 180,E1 4145.726,E2 4145.726} C_VEL
